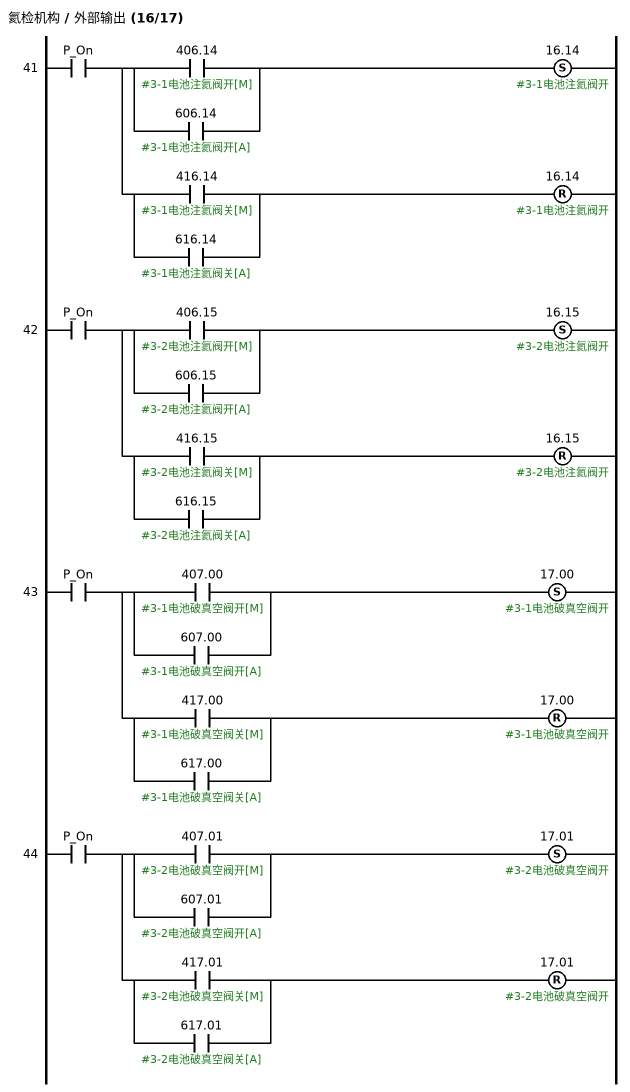
; [picture p384: 氦检机构 / 外部输出, rungs 41-44]
; rung 41
LD P_On
OUT TR0
LD 406.14  ; #3-1电池注氦阀开[M]
OR 606.14  ; #3-1电池注氦阀开[A]
ANDLD
SET 16.14  ; #3-1电池注氦阀开
LD TR0
LD 416.14  ; #3-1电池注氦阀关[M]
OR 616.14  ; #3-1电池注氦阀关[A]
ANDLD
RSET 16.14  ; #3-1电池注氦阀开
; rung 42
LD P_On
OUT TR0
LD 406.15  ; #3-2电池注氦阀开[M]
OR 606.15  ; #3-2电池注氦阀开[A]
ANDLD
SET 16.15  ; #3-2电池注氦阀开
LD TR0
LD 416.15  ; #3-2电池注氦阀关[M]
OR 616.15  ; #3-2电池注氦阀关[A]
ANDLD
RSET 16.15  ; #3-2电池注氦阀开
; rung 43
LD P_On
OUT TR0
LD 407.00  ; #3-1电池破真空阀开[M]
OR 607.00  ; #3-1电池破真空阀开[A]
ANDLD
SET 17.00  ; #3-1电池破真空阀开
LD TR0
LD 417.00  ; #3-1电池破真空阀关[M]
OR 617.00  ; #3-1电池破真空阀关[A]
ANDLD
RSET 17.00  ; #3-1电池破真空阀开
; rung 44
LD P_On
OUT TR0
LD 407.01  ; #3-2电池破真空阀开[M]
OR 607.01  ; #3-2电池破真空阀开[A]
ANDLD
SET 17.01  ; #3-2电池破真空阀开
LD TR0
LD 417.01  ; #3-2电池破真空阀关[M]
OR 617.01  ; #3-2电池破真空阀关[A]
ANDLD
RSET 17.01  ; #3-2电池破真空阀开

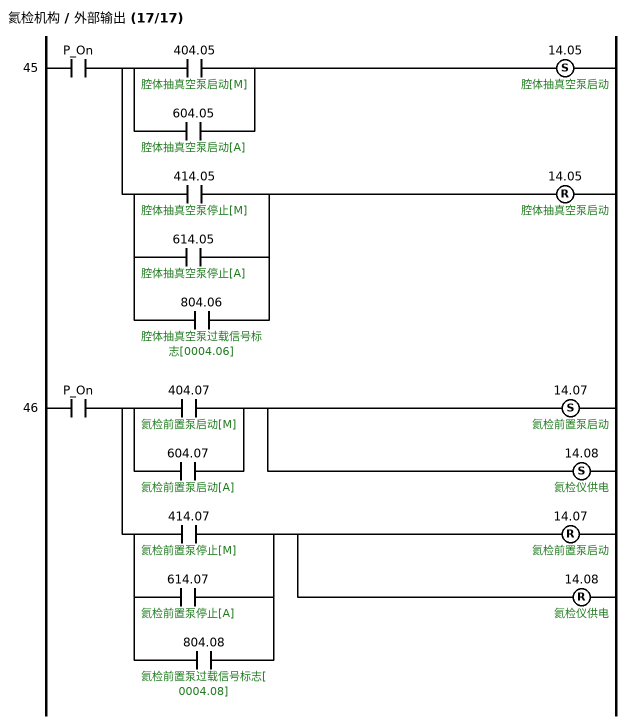
; rung 45
LD P_On
OUT TR0
LD 404.05  ; 腔体抽真空泵启动[M]
OR 604.05  ; 腔体抽真空泵启动[A]
ANDLD
SET 14.05  ; 腔体抽真空泵启动
LD TR0
LD 414.05  ; 腔体抽真空泵停止[M]
OR 614.05  ; 腔体抽真空泵停止[A]
OR 804.06  ; 腔体抽真空泵过载信号标志[0004.06]
ANDLD
RSET 14.05  ; 腔体抽真空泵启动
; rung 46
LD P_On
OUT TR0
LD 404.07  ; 氦检前置泵启动[M]
OR 604.07  ; 氦检前置泵启动[A]
ANDLD
SET 14.07  ; 氦检前置泵启动
SET 14.08  ; 氦检仪供电
LD TR0
LD 414.07  ; 氦检前置泵停止[M]
OR 614.07  ; 氦检前置泵停止[A]
OR 804.08  ; 氦检前置泵过载信号标志[0004.08]
ANDLD
RSET 14.07  ; 氦检前置泵启动
RSET 14.08  ; 氦检仪供电

### Section END
; rung 0
END(001)

## Program 出料伺服机构 (cyclic task 4)

### Section Main

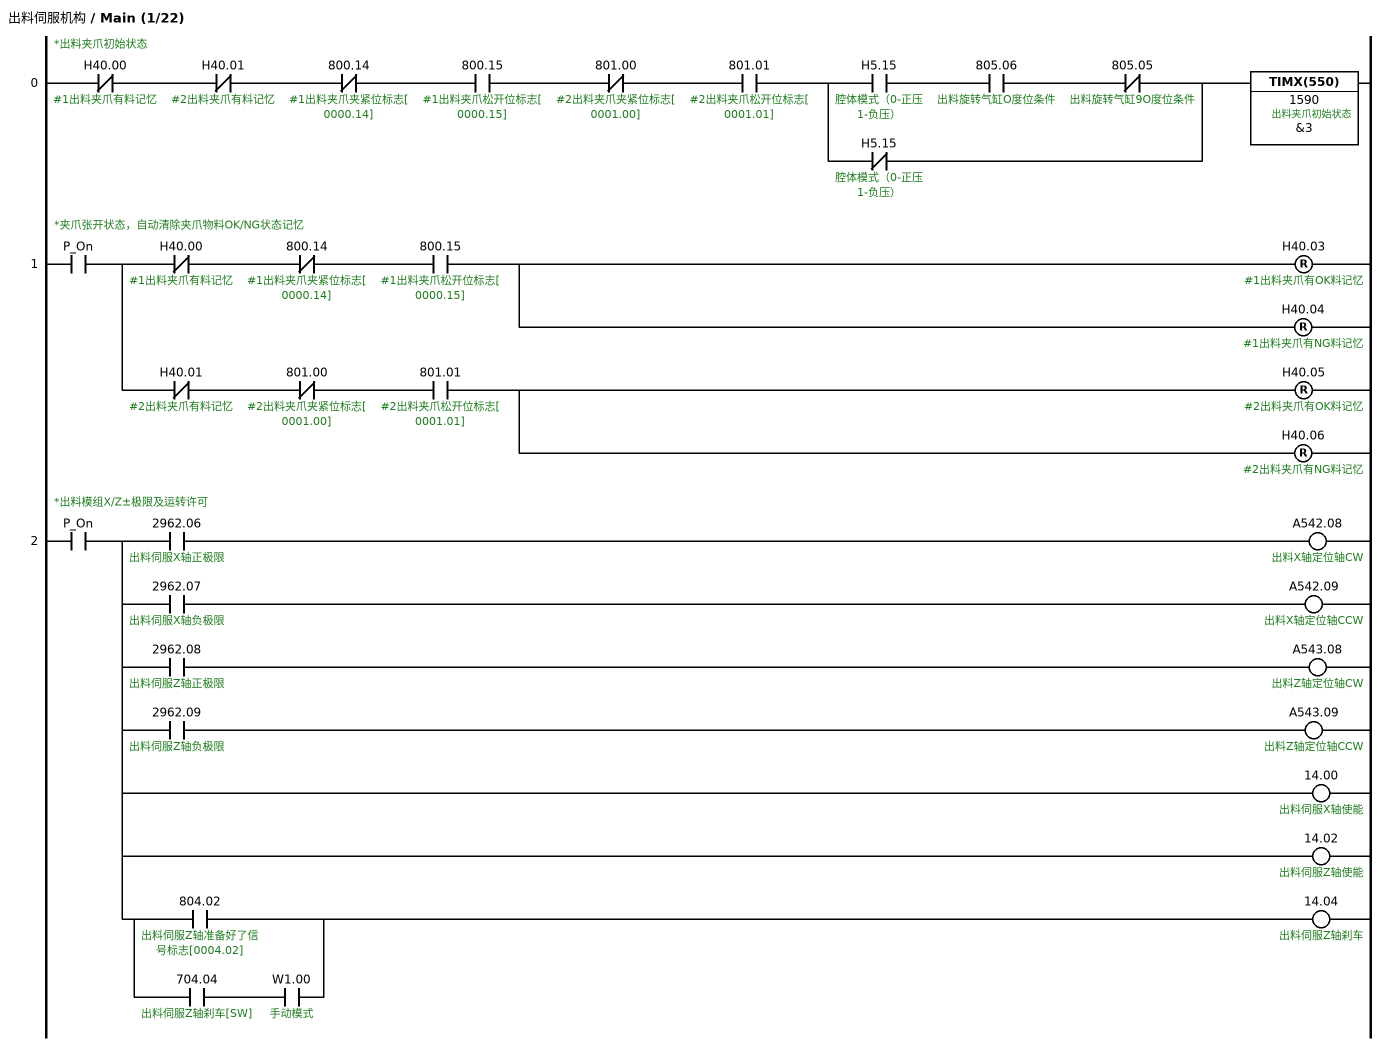
; rung 0: *出料夹爪初始状态
LDNOT H40.00  ; #1出料夹爪有料记忆
ANDNOT H40.01  ; #2出料夹爪有料记忆
ANDNOT 800.14  ; #1出料夹爪夹紧位标志[0000.14]
AND 800.15  ; #1出料夹爪松开位标志[0000.15]
ANDNOT 801.00  ; #2出料夹爪夹紧位标志[0001.00]
AND 801.01  ; #2出料夹爪松开位标志[0001.01]
LD H5.15  ; 腔体模式（0-正压 1-负压）
AND 805.06  ; 出料旋转气缸O度位条件
ANDNOT 805.05  ; 出料旋转气缸9O度位条件
ORNOT H5.15  ; 腔体模式（0-正压 1-负压）
ANDLD
TIMX(550) 1590 &3  ; 出料夹爪初始状态
; rung 1: *夹爪张开状态，自动清除夹爪物料OK/NG状态记忆
LD P_On
OUT TR0
ANDNOT H40.00  ; #1出料夹爪有料记忆
ANDNOT 800.14  ; #1出料夹爪夹紧位标志[0000.14]
AND 800.15  ; #1出料夹爪松开位标志[0000.15]
RSET H40.03  ; #1出料夹爪有OK料记忆
RSET H40.04  ; #1出料夹爪有NG料记忆
LD TR0
ANDNOT H40.01  ; #2出料夹爪有料记忆
ANDNOT 801.00  ; #2出料夹爪夹紧位标志[0001.00]
AND 801.01  ; #2出料夹爪松开位标志[0001.01]
RSET H40.05  ; #2出料夹爪有OK料记忆
RSET H40.06  ; #2出料夹爪有NG料记忆
; rung 2: *出料模组X/Z±极限及运转许可
LD P_On
OUT TR0
AND 2962.06  ; 出料伺服X轴正极限
OUT A542.08  ; 出料X轴定位轴CW
LD TR0
AND 2962.07  ; 出料伺服X轴负极限
OUT A542.09  ; 出料X轴定位轴CCW
LD TR0
AND 2962.08  ; 出料伺服Z轴正极限
OUT A543.08  ; 出料Z轴定位轴CW
LD TR0
AND 2962.09  ; 出料伺服Z轴负极限
OUT A543.09  ; 出料Z轴定位轴CCW
LD TR0
OUT 14.00  ; 出料伺服X轴使能
OUT 14.02  ; 出料伺服Z轴使能
LD 804.02  ; 出料伺服Z轴准备好了信号标志[0004.02]
LD 704.04  ; 出料伺服Z轴刹车[SW]
AND W1.00  ; 手动模式
ORLD
ANDLD
OUT 14.04  ; 出料伺服Z轴刹车

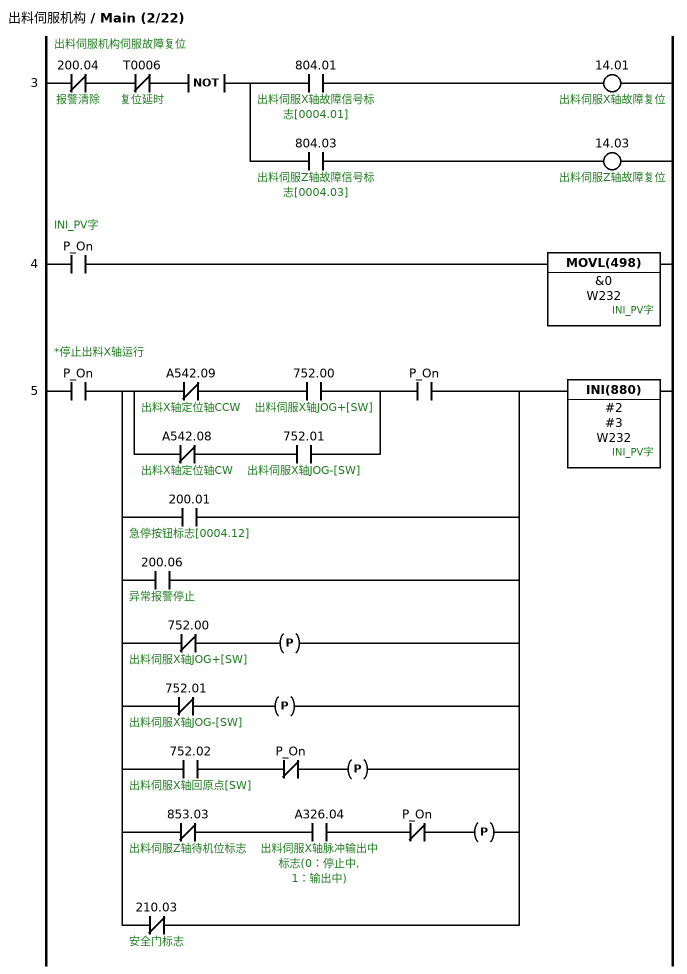
; rung 3: 出料伺服机构伺服故障复位
LDNOT 200.04  ; 报警清除
ANDNOT T0006  ; 复位延时
NOT(520)
OUT TR0
AND 804.01  ; 出料伺服X轴故障信号标志[0004.01]
OUT 14.01  ; 出料伺服X轴故障复位
LD TR0
AND 804.03  ; 出料伺服Z轴故障信号标志[0004.03]
OUT 14.03  ; 出料伺服Z轴故障复位
; rung 4: INI_PV字
LD P_On
MOVL(498) &0 W232  ; INI_PV字
; rung 5: *停止出料X轴运行
LD P_On
LDNOT A542.09  ; 出料X轴定位轴CCW
AND 752.00  ; 出料伺服X轴JOG+[SW]
LDNOT A542.08  ; 出料X轴定位轴CW
AND 752.01  ; 出料伺服X轴JOG-[SW]
ORLD
AND P_On
OR 200.01  ; 急停按钮标志[0004.12]
OR 200.06  ; 异常报警停止
LDNOT 752.00  ; 出料伺服X轴JOG+[SW]
UP(521)
ORLD
LDNOT 752.01  ; 出料伺服X轴JOG-[SW]
UP(521)
ORLD
LD 752.02  ; 出料伺服X轴回原点[SW]
ANDNOT P_On
UP(521)
ORLD
LDNOT 853.03  ; 出料伺服Z轴待机位标志
AND A326.04  ; 出料伺服X轴脉冲输出中标志(0：停止中,1：输出中)
ANDNOT P_On
UP(521)
ORLD
ORNOT 210.03  ; 安全门标志
ANDLD
INI(880) #2 #3 W232  ; INI_PV字

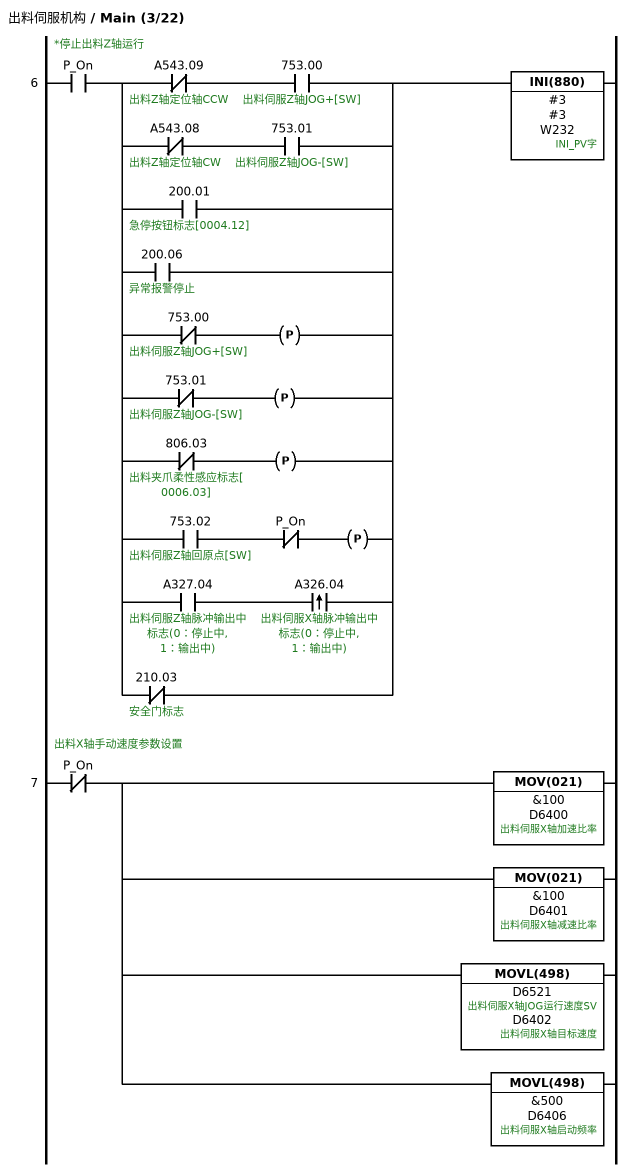
; rung 6: *停止出料Z轴运行
LD P_On
LDNOT A543.09  ; 出料Z轴定位轴CCW
AND 753.00  ; 出料伺服Z轴JOG+[SW]
LDNOT A543.08  ; 出料Z轴定位轴CW
AND 753.01  ; 出料伺服Z轴JOG-[SW]
ORLD
OR 200.01  ; 急停按钮标志[0004.12]
OR 200.06  ; 异常报警停止
LDNOT 753.00  ; 出料伺服Z轴JOG+[SW]
UP(521)
ORLD
LDNOT 753.01  ; 出料伺服Z轴JOG-[SW]
UP(521)
ORLD
LDNOT 806.03  ; 出料夹爪柔性感应标志[0006.03]
UP(521)
ORLD
LD 753.02  ; 出料伺服Z轴回原点[SW]
ANDNOT P_On
UP(521)
ORLD
LD A327.04  ; 出料伺服Z轴脉冲输出中标志(0：停止中,1：输出中)
@AND A326.04  ; 出料伺服X轴脉冲输出中标志(0：停止中,1：输出中)
ORNOT 210.03  ; 安全门标志
ORLD
ANDLD
INI(880) #3 #3 W232  ; INI_PV字
; rung 7: 出料X轴手动速度参数设置
LDNOT P_On
MOV(021) &100 D6400  ; 出料伺服X轴加速比率
MOV(021) &100 D6401  ; 出料伺服X轴减速比率
MOVL(498) D6521 D6402  ; 出料伺服X轴JOG运行速度SV, 出料伺服X轴目标速度
MOVL(498) &500 D6406  ; 出料伺服X轴启动频率

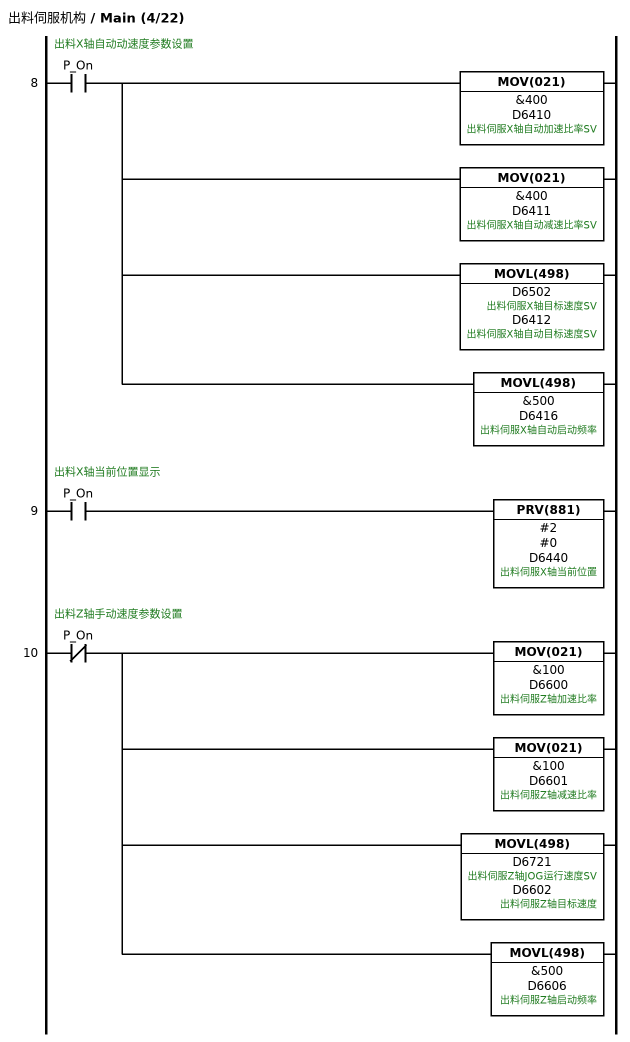
; rung 8: 出料X轴自动动速度参数设置
LD P_On
MOV(021) &400 D6410  ; 出料伺服X轴自动加速比率SV
MOV(021) &400 D6411  ; 出料伺服X轴自动减速比率SV
MOVL(498) D6502 D6412  ; 出料伺服X轴目标速度SV, 出料伺服X轴自动目标速度SV
MOVL(498) &500 D6416  ; 出料伺服X轴自动启动频率
; rung 9: 出料X轴当前位置显示
LD P_On
PRV(881) #2 #0 D6440  ; 出料伺服X轴当前位置
; rung 10: 出料Z轴手动速度参数设置
LDNOT P_On
MOV(021) &100 D6600  ; 出料伺服Z轴加速比率
MOV(021) &100 D6601  ; 出料伺服Z轴减速比率
MOVL(498) D6721 D6602  ; 出料伺服Z轴JOG运行速度SV, 出料伺服Z轴目标速度
MOVL(498) &500 D6606  ; 出料伺服Z轴启动频率

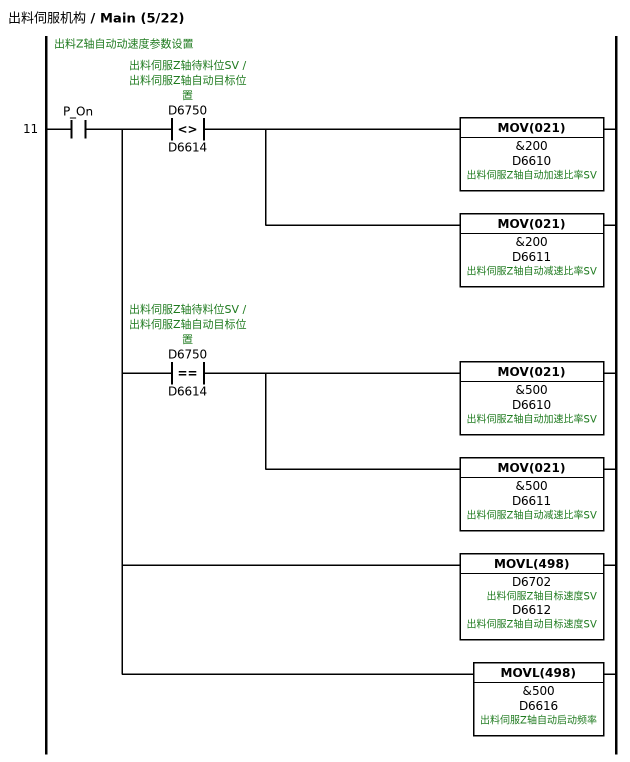
; rung 11: 出料Z轴自动动速度参数设置
LD P_On
OUT TR0
AND<>L(306) D6750 D6614  ; 出料伺服Z轴待料位SV, 出料伺服Z轴自动目标位置
MOV(021) &200 D6610  ; 出料伺服Z轴自动加速比率SV
MOV(021) &200 D6611  ; 出料伺服Z轴自动减速比率SV
LD TR0
AND=L(301) D6750 D6614  ; 出料伺服Z轴待料位SV, 出料伺服Z轴自动目标位置
MOV(021) &500 D6610  ; 出料伺服Z轴自动加速比率SV
MOV(021) &500 D6611  ; 出料伺服Z轴自动减速比率SV
LD TR0
MOVL(498) D6702 D6612  ; 出料伺服Z轴目标速度SV, 出料伺服Z轴自动目标速度SV
MOVL(498) &500 D6616  ; 出料伺服Z轴自动启动频率

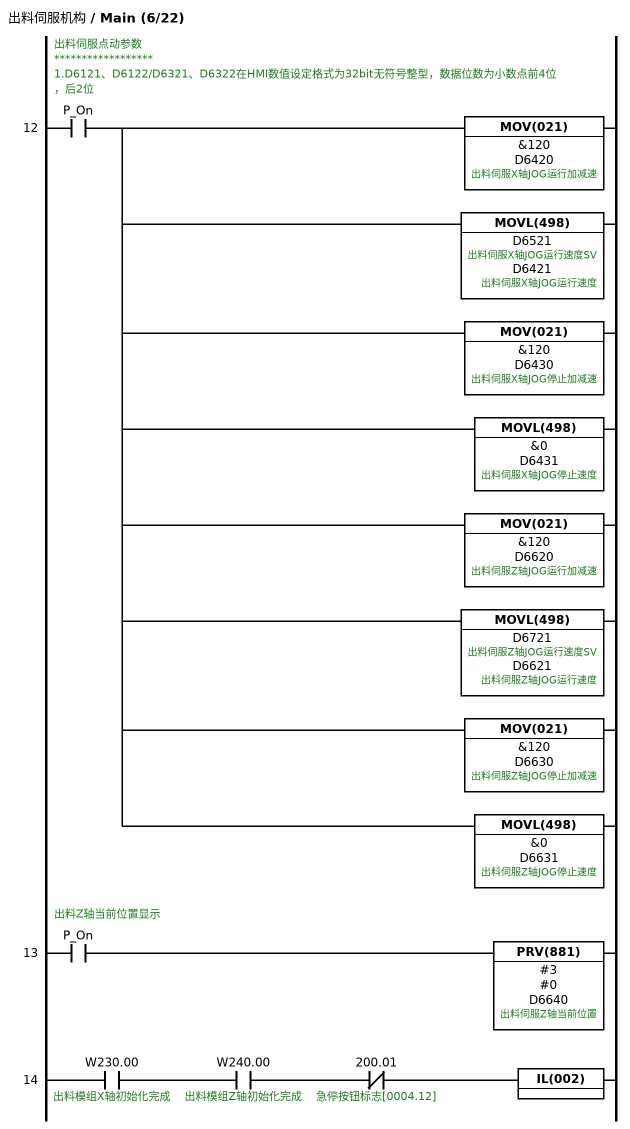
; rung 12: 出料伺服点动参数 / ****************** / 1.D6121、D6122/D6321、D6322在HMI数值设定格式为32bit无符号整型，数据位数为小数点前4位，后2位
LD P_On
MOV(021) &120 D6420  ; 出料伺服X轴JOG运行加减速
MOVL(498) D6521 D6421  ; 出料伺服X轴JOG运行速度SV, 出料伺服X轴JOG运行速度
MOV(021) &120 D6430  ; 出料伺服X轴JOG停止加减速
MOVL(498) &0 D6431  ; 出料伺服X轴JOG停止速度
MOV(021) &120 D6620  ; 出料伺服Z轴JOG运行加减速
MOVL(498) D6721 D6621  ; 出料伺服Z轴JOG运行速度SV, 出料伺服Z轴JOG运行速度
MOV(021) &120 D6630  ; 出料伺服Z轴JOG停止加减速
MOVL(498) &0 D6631  ; 出料伺服Z轴JOG停止速度
; rung 13: 出料Z轴当前位置显示
LD P_On
PRV(881) #3 #0 D6640  ; 出料伺服Z轴当前位置
; rung 14
LD W230.00  ; 出料模组X轴初始化完成
AND W240.00  ; 出料模组Z轴初始化完成
ANDNOT 200.01  ; 急停按钮标志[0004.12]
IL(002)

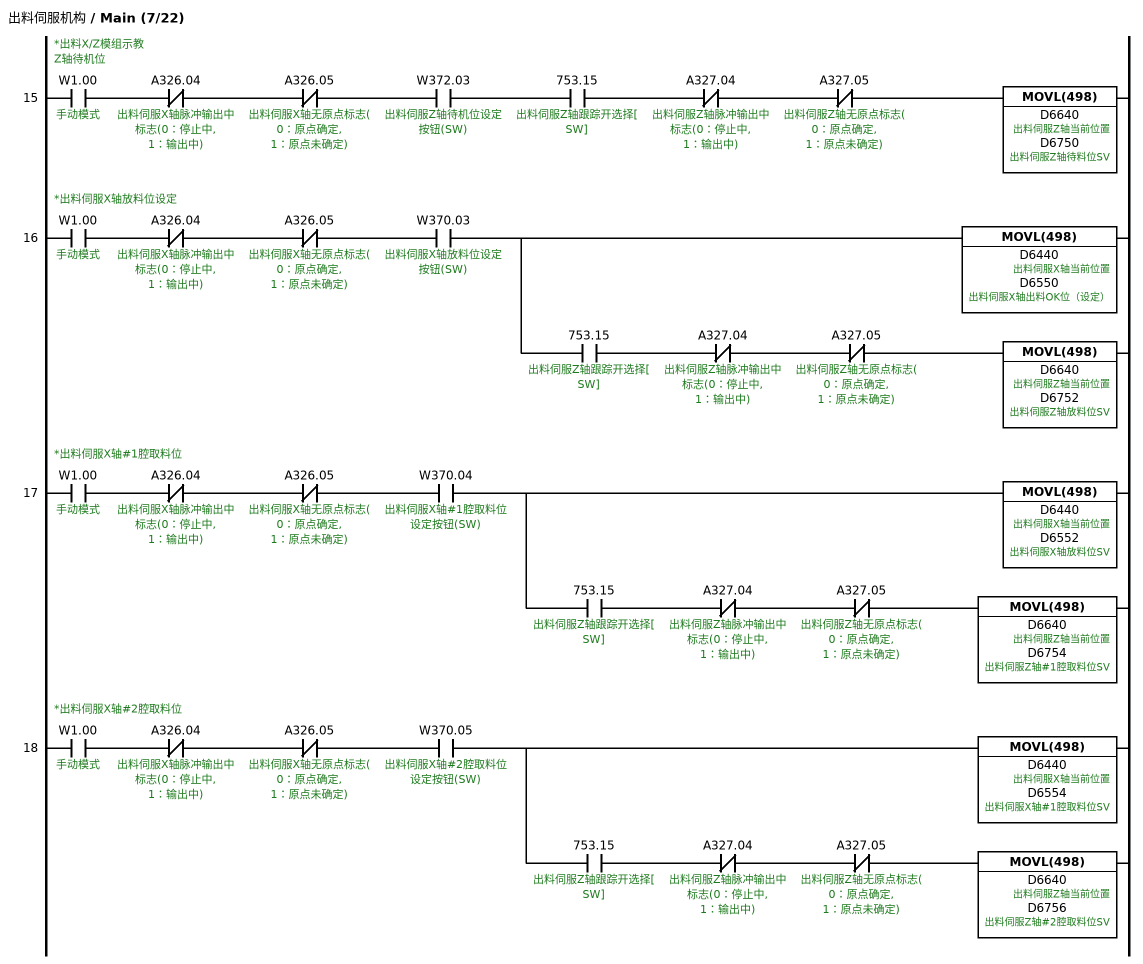
; rung 15: *出料X/Z模组示教 / Z轴待机位
LD W1.00  ; 手动模式
ANDNOT A326.04  ; 出料伺服X轴脉冲输出中标志(0：停止中,1：输出中)
ANDNOT A326.05  ; 出料伺服X轴无原点标志(0：原点确定,1：原点未确定)
AND W372.03  ; 出料伺服Z轴待机位设定按钮(SW)
AND 753.15  ; 出料伺服Z轴跟踪开选择[SW]
ANDNOT A327.04  ; 出料伺服Z轴脉冲输出中标志(0：停止中,1：输出中)
ANDNOT A327.05  ; 出料伺服Z轴无原点标志(0：原点确定,1：原点未确定)
MOVL(498) D6640 D6750  ; 出料伺服Z轴当前位置, 出料伺服Z轴待料位SV
; rung 16: *出料伺服X轴放料位设定
LD W1.00  ; 手动模式
ANDNOT A326.04  ; 出料伺服X轴脉冲输出中标志(0：停止中,1：输出中)
ANDNOT A326.05  ; 出料伺服X轴无原点标志(0：原点确定,1：原点未确定)
AND W370.03  ; 出料伺服X轴放料位设定按钮(SW)
MOVL(498) D6440 D6550  ; 出料伺服X轴当前位置, 出料伺服X轴出料OK位（设定）
AND 753.15  ; 出料伺服Z轴跟踪开选择[SW]
ANDNOT A327.04  ; 出料伺服Z轴脉冲输出中标志(0：停止中,1：输出中)
ANDNOT A327.05  ; 出料伺服Z轴无原点标志(0：原点确定,1：原点未确定)
MOVL(498) D6640 D6752  ; 出料伺服Z轴当前位置, 出料伺服Z轴放料位SV
; rung 17: *出料伺服X轴#1腔取料位
LD W1.00  ; 手动模式
ANDNOT A326.04  ; 出料伺服X轴脉冲输出中标志(0：停止中,1：输出中)
ANDNOT A326.05  ; 出料伺服X轴无原点标志(0：原点确定,1：原点未确定)
AND W370.04  ; 出料伺服X轴#1腔取料位设定按钮(SW)
MOVL(498) D6440 D6552  ; 出料伺服X轴当前位置, 出料伺服X轴放料位SV
AND 753.15  ; 出料伺服Z轴跟踪开选择[SW]
ANDNOT A327.04  ; 出料伺服Z轴脉冲输出中标志(0：停止中,1：输出中)
ANDNOT A327.05  ; 出料伺服Z轴无原点标志(0：原点确定,1：原点未确定)
MOVL(498) D6640 D6754  ; 出料伺服Z轴当前位置, 出料伺服Z轴#1腔取料位SV
; rung 18: *出料伺服X轴#2腔取料位
LD W1.00  ; 手动模式
ANDNOT A326.04  ; 出料伺服X轴脉冲输出中标志(0：停止中,1：输出中)
ANDNOT A326.05  ; 出料伺服X轴无原点标志(0：原点确定,1：原点未确定)
AND W370.05  ; 出料伺服X轴#2腔取料位设定按钮(SW)
MOVL(498) D6440 D6554  ; 出料伺服X轴当前位置, 出料伺服X轴#1腔取料位SV
AND 753.15  ; 出料伺服Z轴跟踪开选择[SW]
ANDNOT A327.04  ; 出料伺服Z轴脉冲输出中标志(0：停止中,1：输出中)
ANDNOT A327.05  ; 出料伺服Z轴无原点标志(0：原点确定,1：原点未确定)
MOVL(498) D6640 D6756  ; 出料伺服Z轴当前位置, 出料伺服Z轴#2腔取料位SV

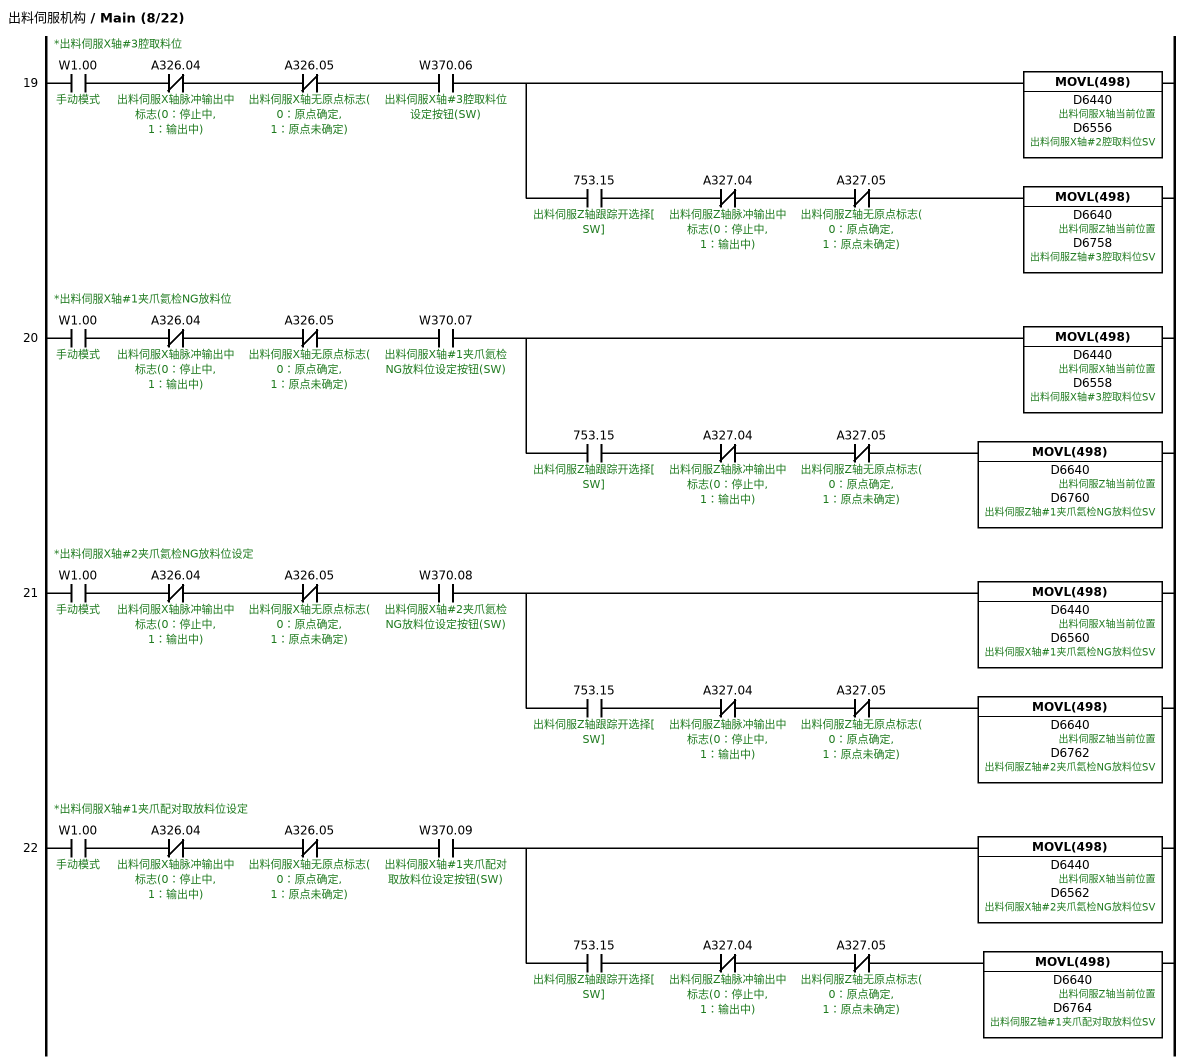
; rung 19: *出料伺服X轴#3腔取料位
LD W1.00  ; 手动模式
ANDNOT A326.04  ; 出料伺服X轴脉冲输出中标志(0：停止中,1：输出中)
ANDNOT A326.05  ; 出料伺服X轴无原点标志(0：原点确定,1：原点未确定)
AND W370.06  ; 出料伺服X轴#3腔取料位设定按钮(SW)
MOVL(498) D6440 D6556  ; 出料伺服X轴当前位置, 出料伺服X轴#2腔取料位SV
AND 753.15  ; 出料伺服Z轴跟踪开选择[SW]
ANDNOT A327.04  ; 出料伺服Z轴脉冲输出中标志(0：停止中,1：输出中)
ANDNOT A327.05  ; 出料伺服Z轴无原点标志(0：原点确定,1：原点未确定)
MOVL(498) D6640 D6758  ; 出料伺服Z轴当前位置, 出料伺服Z轴#3腔取料位SV
; rung 20: *出料伺服X轴#1夹爪氦检NG放料位
LD W1.00  ; 手动模式
ANDNOT A326.04  ; 出料伺服X轴脉冲输出中标志(0：停止中,1：输出中)
ANDNOT A326.05  ; 出料伺服X轴无原点标志(0：原点确定,1：原点未确定)
AND W370.07  ; 出料伺服X轴#1夹爪氦检NG放料位设定按钮(SW)
MOVL(498) D6440 D6558  ; 出料伺服X轴当前位置, 出料伺服X轴#3腔取料位SV
AND 753.15  ; 出料伺服Z轴跟踪开选择[SW]
ANDNOT A327.04  ; 出料伺服Z轴脉冲输出中标志(0：停止中,1：输出中)
ANDNOT A327.05  ; 出料伺服Z轴无原点标志(0：原点确定,1：原点未确定)
MOVL(498) D6640 D6760  ; 出料伺服Z轴当前位置, 出料伺服Z轴#1夹爪氦检NG放料位SV
; rung 21: *出料伺服X轴#2夹爪氦检NG放料位设定
LD W1.00  ; 手动模式
ANDNOT A326.04  ; 出料伺服X轴脉冲输出中标志(0：停止中,1：输出中)
ANDNOT A326.05  ; 出料伺服X轴无原点标志(0：原点确定,1：原点未确定)
AND W370.08  ; 出料伺服X轴#2夹爪氦检NG放料位设定按钮(SW)
MOVL(498) D6440 D6560  ; 出料伺服X轴当前位置, 出料伺服X轴#1夹爪氦检NG放料位SV
AND 753.15  ; 出料伺服Z轴跟踪开选择[SW]
ANDNOT A327.04  ; 出料伺服Z轴脉冲输出中标志(0：停止中,1：输出中)
ANDNOT A327.05  ; 出料伺服Z轴无原点标志(0：原点确定,1：原点未确定)
MOVL(498) D6640 D6762  ; 出料伺服Z轴当前位置, 出料伺服Z轴#2夹爪氦检NG放料位SV
; rung 22: *出料伺服X轴#1夹爪配对取放料位设定
LD W1.00  ; 手动模式
ANDNOT A326.04  ; 出料伺服X轴脉冲输出中标志(0：停止中,1：输出中)
ANDNOT A326.05  ; 出料伺服X轴无原点标志(0：原点确定,1：原点未确定)
AND W370.09  ; 出料伺服X轴#1夹爪配对取放料位设定按钮(SW)
MOVL(498) D6440 D6562  ; 出料伺服X轴当前位置, 出料伺服X轴#2夹爪氦检NG放料位SV
AND 753.15  ; 出料伺服Z轴跟踪开选择[SW]
ANDNOT A327.04  ; 出料伺服Z轴脉冲输出中标志(0：停止中,1：输出中)
ANDNOT A327.05  ; 出料伺服Z轴无原点标志(0：原点确定,1：原点未确定)
MOVL(498) D6640 D6764  ; 出料伺服Z轴当前位置, 出料伺服Z轴#1夹爪配对取放料位SV

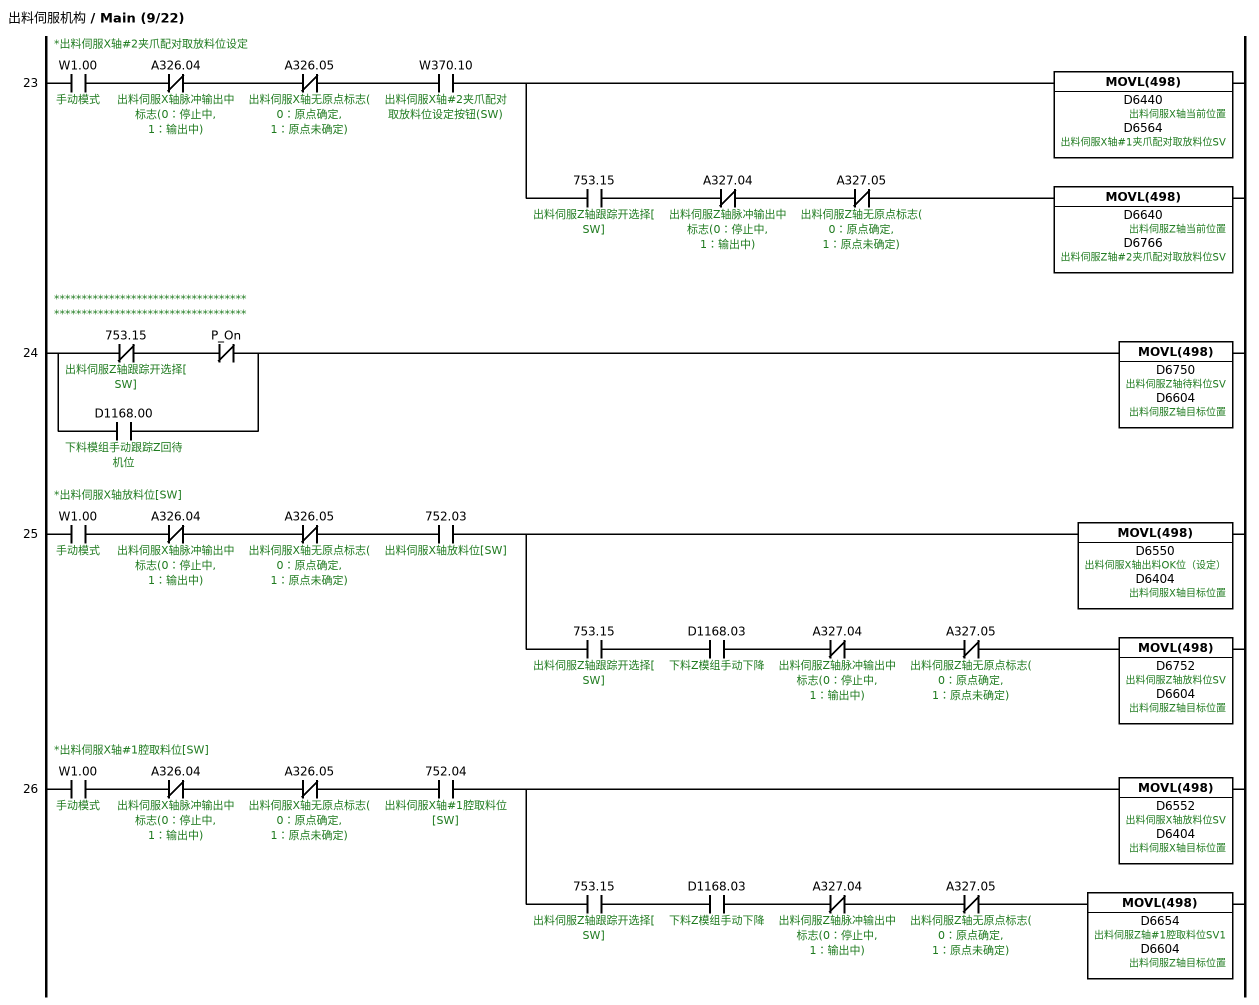
; rung 23: *出料伺服X轴#2夹爪配对取放料位设定
LD W1.00  ; 手动模式
ANDNOT A326.04  ; 出料伺服X轴脉冲输出中标志(0：停止中,1：输出中)
ANDNOT A326.05  ; 出料伺服X轴无原点标志(0：原点确定,1：原点未确定)
AND W370.10  ; 出料伺服X轴#2夹爪配对取放料位设定按钮(SW)
MOVL(498) D6440 D6564  ; 出料伺服X轴当前位置, 出料伺服X轴#1夹爪配对取放料位SV
AND 753.15  ; 出料伺服Z轴跟踪开选择[SW]
ANDNOT A327.04  ; 出料伺服Z轴脉冲输出中标志(0：停止中,1：输出中)
ANDNOT A327.05  ; 出料伺服Z轴无原点标志(0：原点确定,1：原点未确定)
MOVL(498) D6640 D6766  ; 出料伺服Z轴当前位置, 出料伺服Z轴#2夹爪配对取放料位SV
; rung 24: *********************************** / ***********************************
LDNOT 753.15  ; 出料伺服Z轴跟踪开选择[SW]
ANDNOT P_On
OR D1168.00  ; 下料模组手动跟踪Z回待机位
MOVL(498) D6750 D6604  ; 出料伺服Z轴待料位SV, 出料伺服Z轴目标位置
; rung 25: *出料伺服X轴放料位[SW]
LD W1.00  ; 手动模式
ANDNOT A326.04  ; 出料伺服X轴脉冲输出中标志(0：停止中,1：输出中)
ANDNOT A326.05  ; 出料伺服X轴无原点标志(0：原点确定,1：原点未确定)
AND 752.03  ; 出料伺服X轴放料位[SW]
MOVL(498) D6550 D6404  ; 出料伺服X轴出料OK位（设定）, 出料伺服X轴目标位置
AND 753.15  ; 出料伺服Z轴跟踪开选择[SW]
AND D1168.03  ; 下料Z模组手动下降
ANDNOT A327.04  ; 出料伺服Z轴脉冲输出中标志(0：停止中,1：输出中)
ANDNOT A327.05  ; 出料伺服Z轴无原点标志(0：原点确定,1：原点未确定)
MOVL(498) D6752 D6604  ; 出料伺服Z轴放料位SV, 出料伺服Z轴目标位置
; rung 26: *出料伺服X轴#1腔取料位[SW]
LD W1.00  ; 手动模式
ANDNOT A326.04  ; 出料伺服X轴脉冲输出中标志(0：停止中,1：输出中)
ANDNOT A326.05  ; 出料伺服X轴无原点标志(0：原点确定,1：原点未确定)
AND 752.04  ; 出料伺服X轴#1腔取料位[SW]
MOVL(498) D6552 D6404  ; 出料伺服X轴放料位SV, 出料伺服X轴目标位置
AND 753.15  ; 出料伺服Z轴跟踪开选择[SW]
AND D1168.03  ; 下料Z模组手动下降
ANDNOT A327.04  ; 出料伺服Z轴脉冲输出中标志(0：停止中,1：输出中)
ANDNOT A327.05  ; 出料伺服Z轴无原点标志(0：原点确定,1：原点未确定)
MOVL(498) D6654 D6604  ; 出料伺服Z轴#1腔取料位SV1, 出料伺服Z轴目标位置

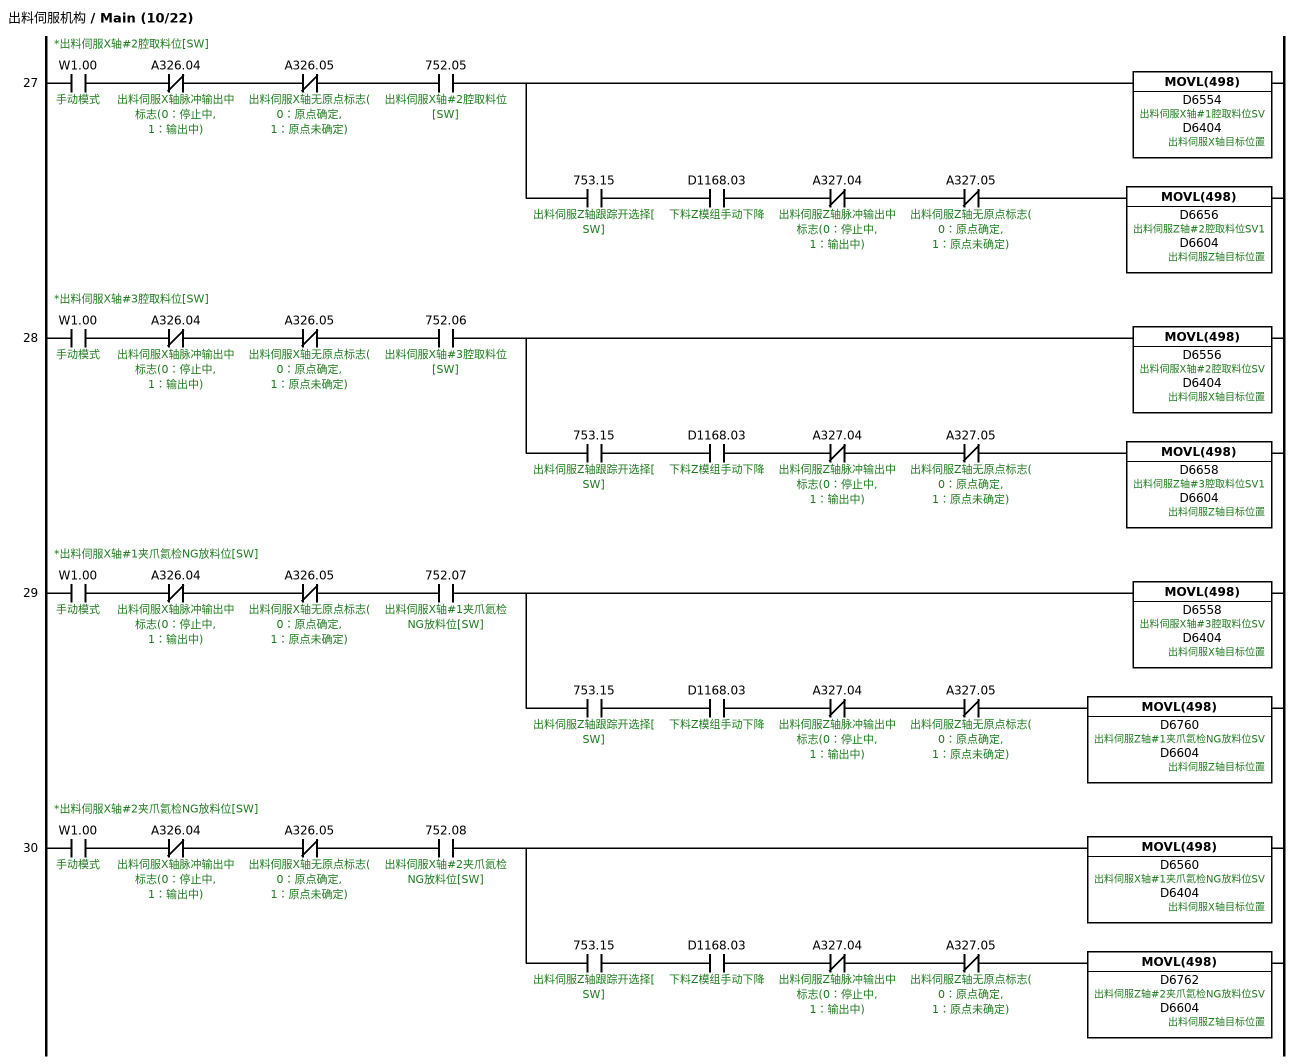
; rung 27: *出料伺服X轴#2腔取料位[SW]
LD W1.00  ; 手动模式
ANDNOT A326.04  ; 出料伺服X轴脉冲输出中标志(0：停止中,1：输出中)
ANDNOT A326.05  ; 出料伺服X轴无原点标志(0：原点确定,1：原点未确定)
AND 752.05  ; 出料伺服X轴#2腔取料位[SW]
MOVL(498) D6554 D6404  ; 出料伺服X轴#1腔取料位SV, 出料伺服X轴目标位置
AND 753.15  ; 出料伺服Z轴跟踪开选择[SW]
AND D1168.03  ; 下料Z模组手动下降
ANDNOT A327.04  ; 出料伺服Z轴脉冲输出中标志(0：停止中,1：输出中)
ANDNOT A327.05  ; 出料伺服Z轴无原点标志(0：原点确定,1：原点未确定)
MOVL(498) D6656 D6604  ; 出料伺服Z轴#2腔取料位SV1, 出料伺服Z轴目标位置
; rung 28: *出料伺服X轴#3腔取料位[SW]
LD W1.00  ; 手动模式
ANDNOT A326.04  ; 出料伺服X轴脉冲输出中标志(0：停止中,1：输出中)
ANDNOT A326.05  ; 出料伺服X轴无原点标志(0：原点确定,1：原点未确定)
AND 752.06  ; 出料伺服X轴#3腔取料位[SW]
MOVL(498) D6556 D6404  ; 出料伺服X轴#2腔取料位SV, 出料伺服X轴目标位置
AND 753.15  ; 出料伺服Z轴跟踪开选择[SW]
AND D1168.03  ; 下料Z模组手动下降
ANDNOT A327.04  ; 出料伺服Z轴脉冲输出中标志(0：停止中,1：输出中)
ANDNOT A327.05  ; 出料伺服Z轴无原点标志(0：原点确定,1：原点未确定)
MOVL(498) D6658 D6604  ; 出料伺服Z轴#3腔取料位SV1, 出料伺服Z轴目标位置
; rung 29: *出料伺服X轴#1夹爪氦检NG放料位[SW]
LD W1.00  ; 手动模式
ANDNOT A326.04  ; 出料伺服X轴脉冲输出中标志(0：停止中,1：输出中)
ANDNOT A326.05  ; 出料伺服X轴无原点标志(0：原点确定,1：原点未确定)
AND 752.07  ; 出料伺服X轴#1夹爪氦检NG放料位[SW]
MOVL(498) D6558 D6404  ; 出料伺服X轴#3腔取料位SV, 出料伺服X轴目标位置
AND 753.15  ; 出料伺服Z轴跟踪开选择[SW]
AND D1168.03  ; 下料Z模组手动下降
ANDNOT A327.04  ; 出料伺服Z轴脉冲输出中标志(0：停止中,1：输出中)
ANDNOT A327.05  ; 出料伺服Z轴无原点标志(0：原点确定,1：原点未确定)
MOVL(498) D6760 D6604  ; 出料伺服Z轴#1夹爪氦检NG放料位SV, 出料伺服Z轴目标位置
; rung 30: *出料伺服X轴#2夹爪氦检NG放料位[SW]
LD W1.00  ; 手动模式
ANDNOT A326.04  ; 出料伺服X轴脉冲输出中标志(0：停止中,1：输出中)
ANDNOT A326.05  ; 出料伺服X轴无原点标志(0：原点确定,1：原点未确定)
AND 752.08  ; 出料伺服X轴#2夹爪氦检NG放料位[SW]
MOVL(498) D6560 D6404  ; 出料伺服X轴#1夹爪氦检NG放料位SV, 出料伺服X轴目标位置
AND 753.15  ; 出料伺服Z轴跟踪开选择[SW]
AND D1168.03  ; 下料Z模组手动下降
ANDNOT A327.04  ; 出料伺服Z轴脉冲输出中标志(0：停止中,1：输出中)
ANDNOT A327.05  ; 出料伺服Z轴无原点标志(0：原点确定,1：原点未确定)
MOVL(498) D6762 D6604  ; 出料伺服Z轴#2夹爪氦检NG放料位SV, 出料伺服Z轴目标位置

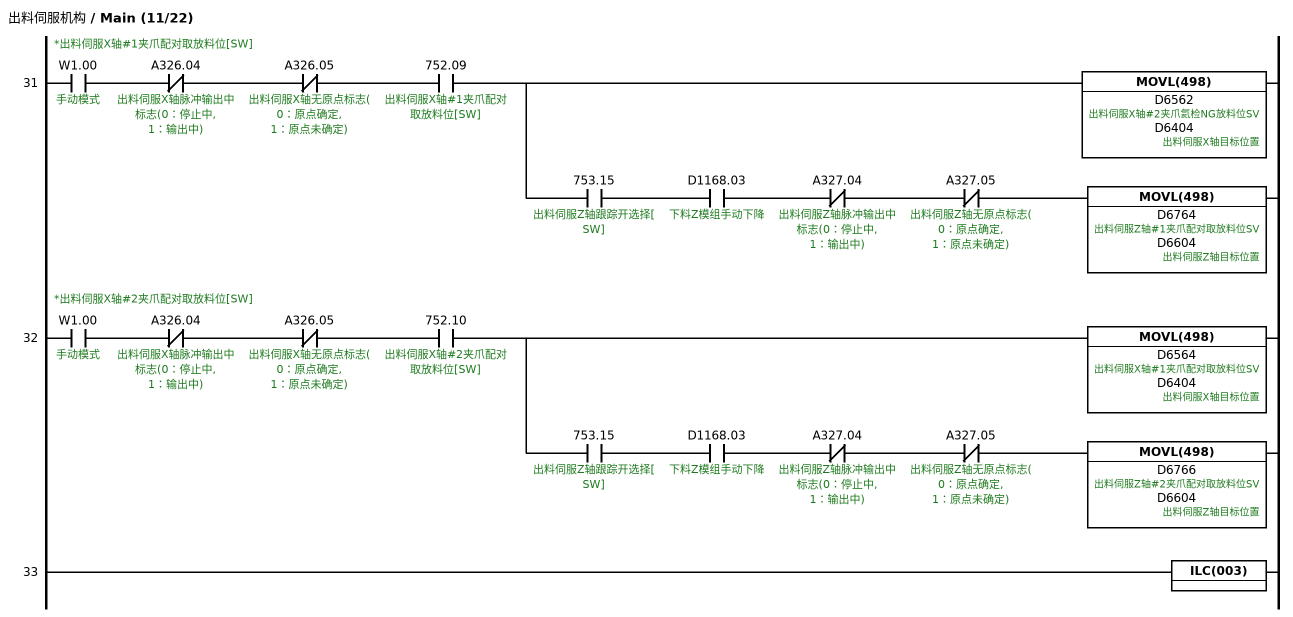
; rung 31: *出料伺服X轴#1夹爪配对取放料位[SW]
LD W1.00  ; 手动模式
ANDNOT A326.04  ; 出料伺服X轴脉冲输出中标志(0：停止中,1：输出中)
ANDNOT A326.05  ; 出料伺服X轴无原点标志(0：原点确定,1：原点未确定)
AND 752.09  ; 出料伺服X轴#1夹爪配对取放料位[SW]
MOVL(498) D6562 D6404  ; 出料伺服X轴#2夹爪氦检NG放料位SV, 出料伺服X轴目标位置
AND 753.15  ; 出料伺服Z轴跟踪开选择[SW]
AND D1168.03  ; 下料Z模组手动下降
ANDNOT A327.04  ; 出料伺服Z轴脉冲输出中标志(0：停止中,1：输出中)
ANDNOT A327.05  ; 出料伺服Z轴无原点标志(0：原点确定,1：原点未确定)
MOVL(498) D6764 D6604  ; 出料伺服Z轴#1夹爪配对取放料位SV, 出料伺服Z轴目标位置
; rung 32: *出料伺服X轴#2夹爪配对取放料位[SW]
LD W1.00  ; 手动模式
ANDNOT A326.04  ; 出料伺服X轴脉冲输出中标志(0：停止中,1：输出中)
ANDNOT A326.05  ; 出料伺服X轴无原点标志(0：原点确定,1：原点未确定)
AND 752.10  ; 出料伺服X轴#2夹爪配对取放料位[SW]
MOVL(498) D6564 D6404  ; 出料伺服X轴#1夹爪配对取放料位SV, 出料伺服X轴目标位置
AND 753.15  ; 出料伺服Z轴跟踪开选择[SW]
AND D1168.03  ; 下料Z模组手动下降
ANDNOT A327.04  ; 出料伺服Z轴脉冲输出中标志(0：停止中,1：输出中)
ANDNOT A327.05  ; 出料伺服Z轴无原点标志(0：原点确定,1：原点未确定)
MOVL(498) D6766 D6604  ; 出料伺服Z轴#2夹爪配对取放料位SV, 出料伺服Z轴目标位置
; rung 33
ILC(003)

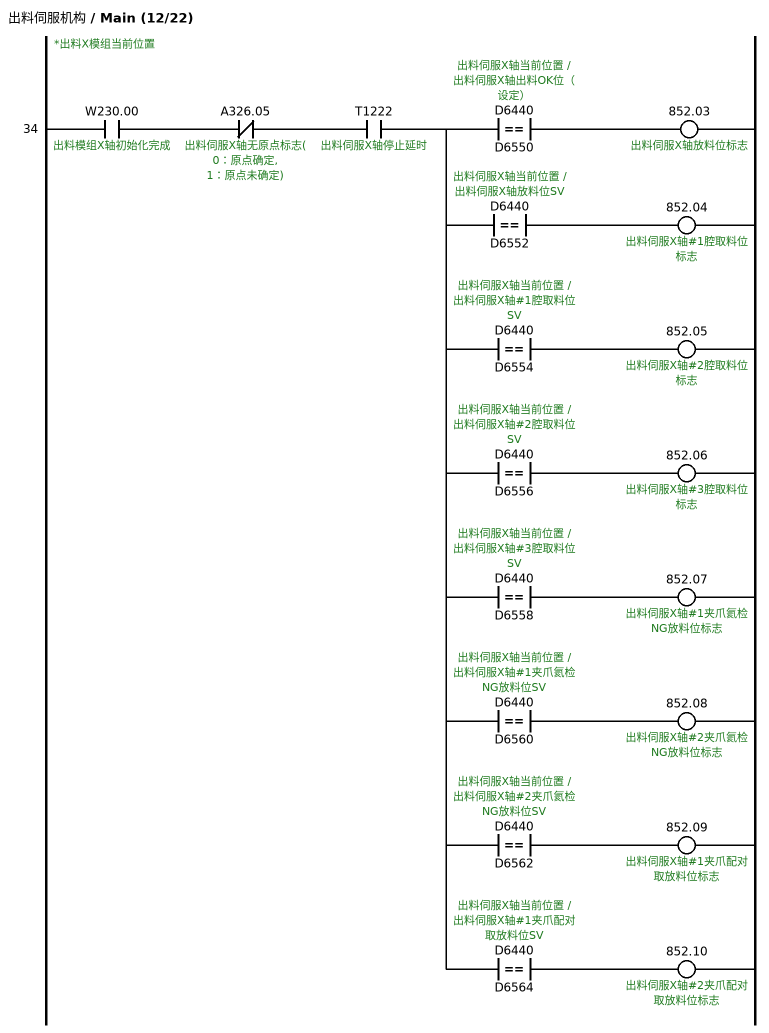
; rung 34: *出料X模组当前位置
LD W230.00  ; 出料模组X轴初始化完成
ANDNOT A326.05  ; 出料伺服X轴无原点标志(0：原点确定,1：原点未确定)
AND T1222  ; 出料伺服X轴停止延时
OUT TR0
AND=SL(303) D6440 D6550  ; 出料伺服X轴当前位置, 出料伺服X轴出料OK位（设定）
OUT 852.03  ; 出料伺服X轴放料位标志
LD TR0
AND=SL(303) D6440 D6552  ; 出料伺服X轴当前位置, 出料伺服X轴放料位SV
OUT 852.04  ; 出料伺服X轴#1腔取料位标志
LD TR0
AND=SL(303) D6440 D6554  ; 出料伺服X轴当前位置, 出料伺服X轴#1腔取料位SV
OUT 852.05  ; 出料伺服X轴#2腔取料位标志
LD TR0
AND=SL(303) D6440 D6556  ; 出料伺服X轴当前位置, 出料伺服X轴#2腔取料位SV
OUT 852.06  ; 出料伺服X轴#3腔取料位标志
LD TR0
AND=SL(303) D6440 D6558  ; 出料伺服X轴当前位置, 出料伺服X轴#3腔取料位SV
OUT 852.07  ; 出料伺服X轴#1夹爪氦检NG放料位标志
LD TR0
AND=SL(303) D6440 D6560  ; 出料伺服X轴当前位置, 出料伺服X轴#1夹爪氦检NG放料位SV
OUT 852.08  ; 出料伺服X轴#2夹爪氦检NG放料位标志
LD TR0
AND=SL(303) D6440 D6562  ; 出料伺服X轴当前位置, 出料伺服X轴#2夹爪氦检NG放料位SV
OUT 852.09  ; 出料伺服X轴#1夹爪配对取放料位标志
LD TR0
AND=SL(303) D6440 D6564  ; 出料伺服X轴当前位置, 出料伺服X轴#1夹爪配对取放料位SV
OUT 852.10  ; 出料伺服X轴#2夹爪配对取放料位标志

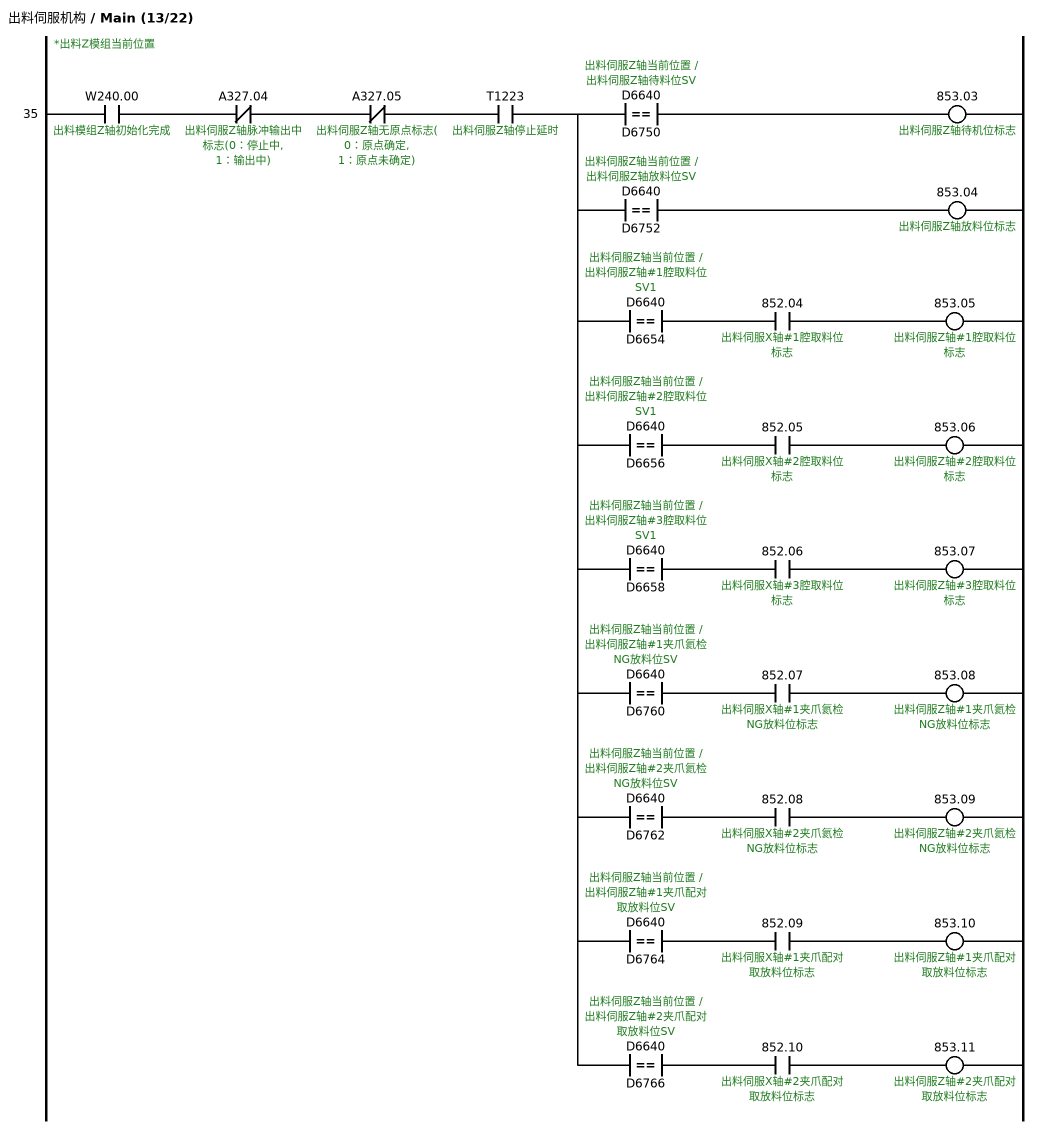
; rung 35: *出料Z模组当前位置
LD W240.00  ; 出料模组Z轴初始化完成
ANDNOT A327.04  ; 出料伺服Z轴脉冲输出中标志(0：停止中,1：输出中)
ANDNOT A327.05  ; 出料伺服Z轴无原点标志(0：原点确定,1：原点未确定)
AND T1223  ; 出料伺服Z轴停止延时
OUT TR0
AND=SL(303) D6640 D6750  ; 出料伺服Z轴当前位置, 出料伺服Z轴待料位SV
OUT 853.03  ; 出料伺服Z轴待机位标志
LD TR0
AND=SL(303) D6640 D6752  ; 出料伺服Z轴当前位置, 出料伺服Z轴放料位SV
OUT 853.04  ; 出料伺服Z轴放料位标志
LD TR0
AND=SL(303) D6640 D6654  ; 出料伺服Z轴当前位置, 出料伺服Z轴#1腔取料位SV1
AND 852.04  ; 出料伺服X轴#1腔取料位标志
OUT 853.05  ; 出料伺服Z轴#1腔取料位标志
LD TR0
AND=SL(303) D6640 D6656  ; 出料伺服Z轴当前位置, 出料伺服Z轴#2腔取料位SV1
AND 852.05  ; 出料伺服X轴#2腔取料位标志
OUT 853.06  ; 出料伺服Z轴#2腔取料位标志
LD TR0
AND=SL(303) D6640 D6658  ; 出料伺服Z轴当前位置, 出料伺服Z轴#3腔取料位SV1
AND 852.06  ; 出料伺服X轴#3腔取料位标志
OUT 853.07  ; 出料伺服Z轴#3腔取料位标志
LD TR0
AND=SL(303) D6640 D6760  ; 出料伺服Z轴当前位置, 出料伺服Z轴#1夹爪氦检NG放料位SV
AND 852.07  ; 出料伺服X轴#1夹爪氦检NG放料位标志
OUT 853.08  ; 出料伺服Z轴#1夹爪氦检NG放料位标志
LD TR0
AND=SL(303) D6640 D6762  ; 出料伺服Z轴当前位置, 出料伺服Z轴#2夹爪氦检NG放料位SV
AND 852.08  ; 出料伺服X轴#2夹爪氦检NG放料位标志
OUT 853.09  ; 出料伺服Z轴#2夹爪氦检NG放料位标志
LD TR0
AND=SL(303) D6640 D6764  ; 出料伺服Z轴当前位置, 出料伺服Z轴#1夹爪配对取放料位SV
AND 852.09  ; 出料伺服X轴#1夹爪配对取放料位标志
OUT 853.10  ; 出料伺服Z轴#1夹爪配对取放料位标志
LD TR0
AND=SL(303) D6640 D6766  ; 出料伺服Z轴当前位置, 出料伺服Z轴#2夹爪配对取放料位SV
AND 852.10  ; 出料伺服X轴#2夹爪配对取放料位标志
OUT 853.11  ; 出料伺服Z轴#2夹爪配对取放料位标志

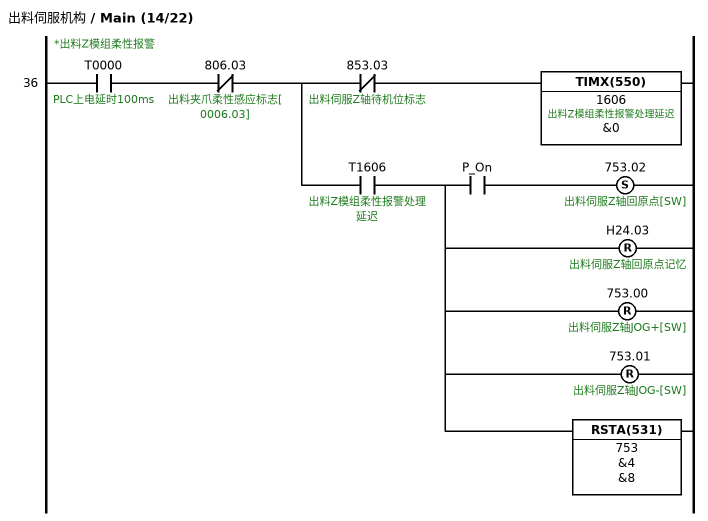
; rung 36: *出料Z模组柔性报警
LD T0000  ; PLC上电延时100ms
ANDNOT 806.03  ; 出料夹爪柔性感应标志[0006.03]
OUT TR0
ANDNOT 853.03  ; 出料伺服Z轴待机位标志
TIMX(550) 1606 &0  ; 出料Z模组柔性报警处理延迟
LD TR0
AND T1606  ; 出料Z模组柔性报警处理延迟
OUT TR0
AND P_On
SET 753.02  ; 出料伺服Z轴回原点[SW]
LD TR0
RSET H24.03  ; 出料伺服Z轴回原点记忆
RSET 753.00  ; 出料伺服Z轴JOG+[SW]
RSET 753.01  ; 出料伺服Z轴JOG-[SW]
RSTA(531) 753 &4 &8

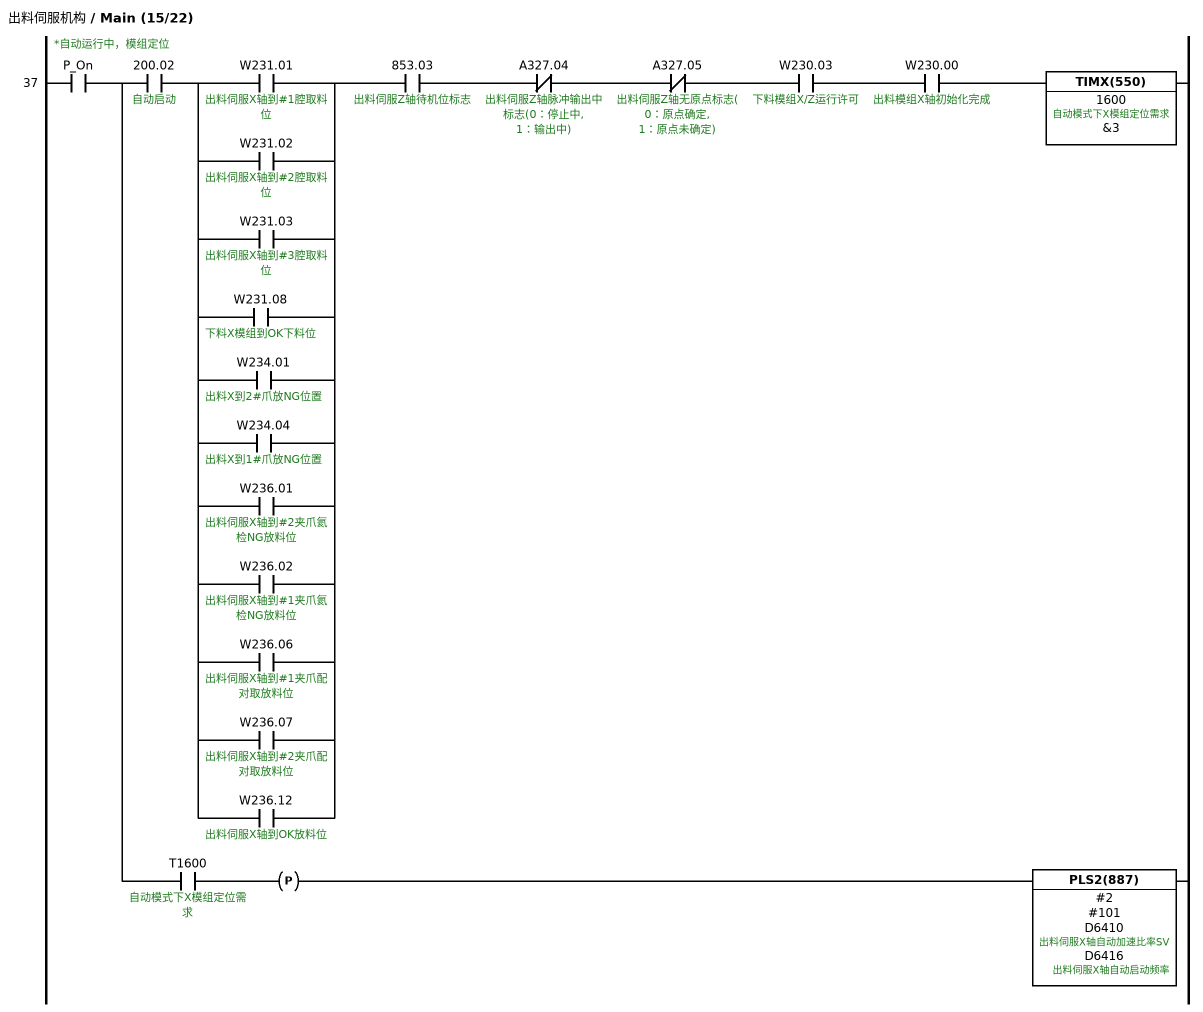
; rung 37: *自动运行中，模组定位
LD P_On
OUT TR0
AND 200.02  ; 自动启动
LD W231.01  ; 出料伺服X轴到#1腔取料位
OR W231.02  ; 出料伺服X轴到#2腔取料位
OR W231.03  ; 出料伺服X轴到#3腔取料位
OR W231.08  ; 下料X模组到OK下料位
OR W234.01  ; 出料X到2#爪放NG位置
OR W234.04  ; 出料X到1#爪放NG位置
OR W236.01  ; 出料伺服X轴到#2夹爪氦检NG放料位
OR W236.02  ; 出料伺服X轴到#1夹爪氦检NG放料位
OR W236.06  ; 出料伺服X轴到#1夹爪配对取放料位
OR W236.07  ; 出料伺服X轴到#2夹爪配对取放料位
OR W236.12  ; 出料伺服X轴到OK放料位
ANDLD
AND 853.03  ; 出料伺服Z轴待机位标志
ANDNOT A327.04  ; 出料伺服Z轴脉冲输出中标志(0：停止中,1：输出中)
ANDNOT A327.05  ; 出料伺服Z轴无原点标志(0：原点确定,1：原点未确定)
AND W230.03  ; 下料模组X/Z运行许可
AND W230.00  ; 出料模组X轴初始化完成
TIMX(550) 1600 &3  ; 自动模式下X模组定位需求
LD TR0
AND T1600  ; 自动模式下X模组定位需求
UP(521)
PLS2(887) #2 #101 D6410 D6416  ; 出料伺服X轴自动加速比率SV, 出料伺服X轴自动启动频率

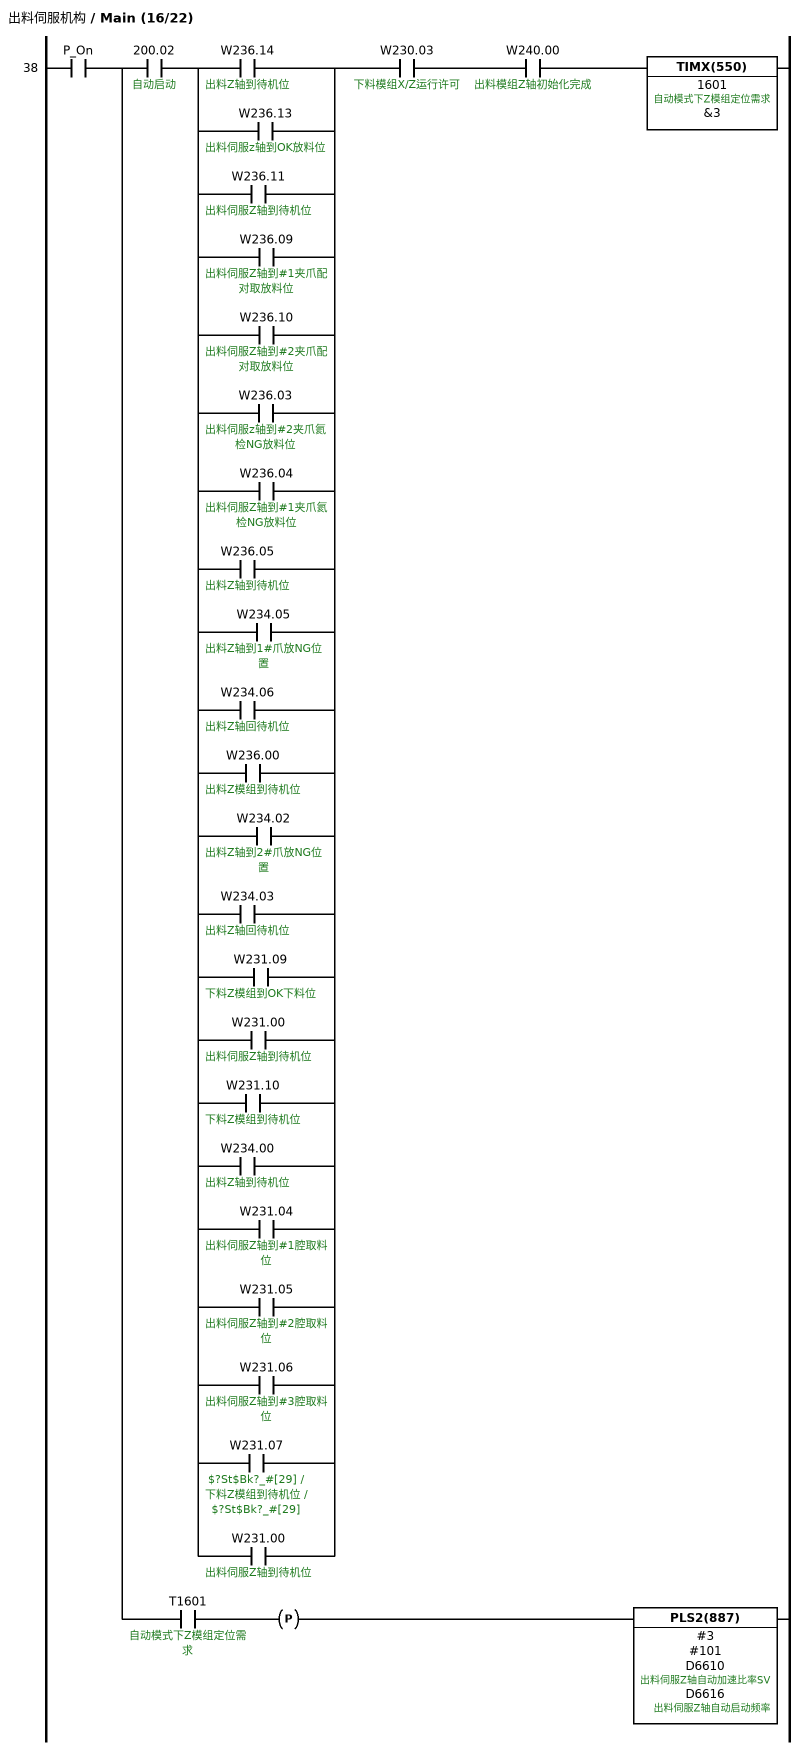
; rung 38
LD P_On
OUT TR0
AND 200.02  ; 自动启动
LD W236.14  ; 出料Z轴到待机位
OR W236.13  ; 出料伺服z轴到OK放料位
OR W236.11  ; 出料伺服Z轴到待机位
OR W236.09  ; 出料伺服Z轴到#1夹爪配对取放料位
OR W236.10  ; 出料伺服Z轴到#2夹爪配对取放料位
OR W236.03  ; 出料伺服z轴到#2夹爪氦检NG放料位
OR W236.04  ; 出料伺服Z轴到#1夹爪氦检NG放料位
OR W236.05  ; 出料Z轴到待机位
OR W234.05  ; 出料Z轴到1#爪放NG位置
OR W234.06  ; 出料Z轴回待机位
OR W236.00  ; 出料Z模组到待机位
OR W234.02  ; 出料Z轴到2#爪放NG位置
OR W234.03  ; 出料Z轴回待机位
OR W231.09  ; 下料Z模组到OK下料位
OR W231.00  ; 出料伺服Z轴到待机位
OR W231.10  ; 下料Z模组到待机位
OR W234.00  ; 出料Z轴到待机位
OR W231.04  ; 出料伺服Z轴到#1腔取料位
OR W231.05  ; 出料伺服Z轴到#2腔取料位
OR W231.06  ; 出料伺服Z轴到#3腔取料位
OR W231.07  ; $?St$Bk?_#[29] / 下料Z模组到待机位 / $?St$Bk?_#[29]
OR W231.00  ; 出料伺服Z轴到待机位
ANDLD
AND W230.03  ; 下料模组X/Z运行许可
AND W240.00  ; 出料模组Z轴初始化完成
TIMX(550) 1601 &3  ; 自动模式下Z模组定位需求
LD TR0
AND T1601  ; 自动模式下Z模组定位需求
UP(521)
PLS2(887) #3 #101 D6610 D6616  ; 出料伺服Z轴自动加速比率SV, 出料伺服Z轴自动启动频率

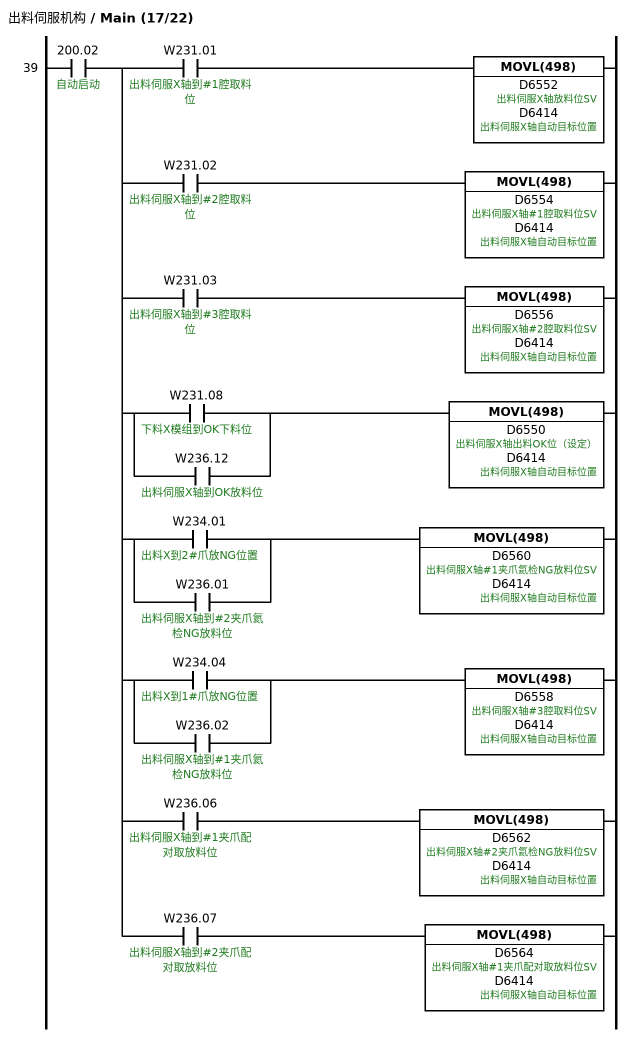
; rung 39
LD 200.02  ; 自动启动
OUT TR0
AND W231.01  ; 出料伺服X轴到#1腔取料位
MOVL(498) D6552 D6414  ; 出料伺服X轴放料位SV, 出料伺服X轴自动目标位置
LD TR0
AND W231.02  ; 出料伺服X轴到#2腔取料位
MOVL(498) D6554 D6414  ; 出料伺服X轴#1腔取料位SV, 出料伺服X轴自动目标位置
LD TR0
AND W231.03  ; 出料伺服X轴到#3腔取料位
MOVL(498) D6556 D6414  ; 出料伺服X轴#2腔取料位SV, 出料伺服X轴自动目标位置
LD TR0
LD W231.08  ; 下料X模组到OK下料位
OR W236.12  ; 出料伺服X轴到OK放料位
ANDLD
MOVL(498) D6550 D6414  ; 出料伺服X轴出料OK位（设定）, 出料伺服X轴自动目标位置
LD TR0
LD W234.01  ; 出料X到2#爪放NG位置
OR W236.01  ; 出料伺服X轴到#2夹爪氦检NG放料位
ANDLD
MOVL(498) D6560 D6414  ; 出料伺服X轴#1夹爪氦检NG放料位SV, 出料伺服X轴自动目标位置
LD TR0
LD W234.04  ; 出料X到1#爪放NG位置
OR W236.02  ; 出料伺服X轴到#1夹爪氦检NG放料位
ANDLD
MOVL(498) D6558 D6414  ; 出料伺服X轴#3腔取料位SV, 出料伺服X轴自动目标位置
LD TR0
AND W236.06  ; 出料伺服X轴到#1夹爪配对取放料位
MOVL(498) D6562 D6414  ; 出料伺服X轴#2夹爪氦检NG放料位SV, 出料伺服X轴自动目标位置
LD TR0
AND W236.07  ; 出料伺服X轴到#2夹爪配对取放料位
MOVL(498) D6564 D6414  ; 出料伺服X轴#1夹爪配对取放料位SV, 出料伺服X轴自动目标位置

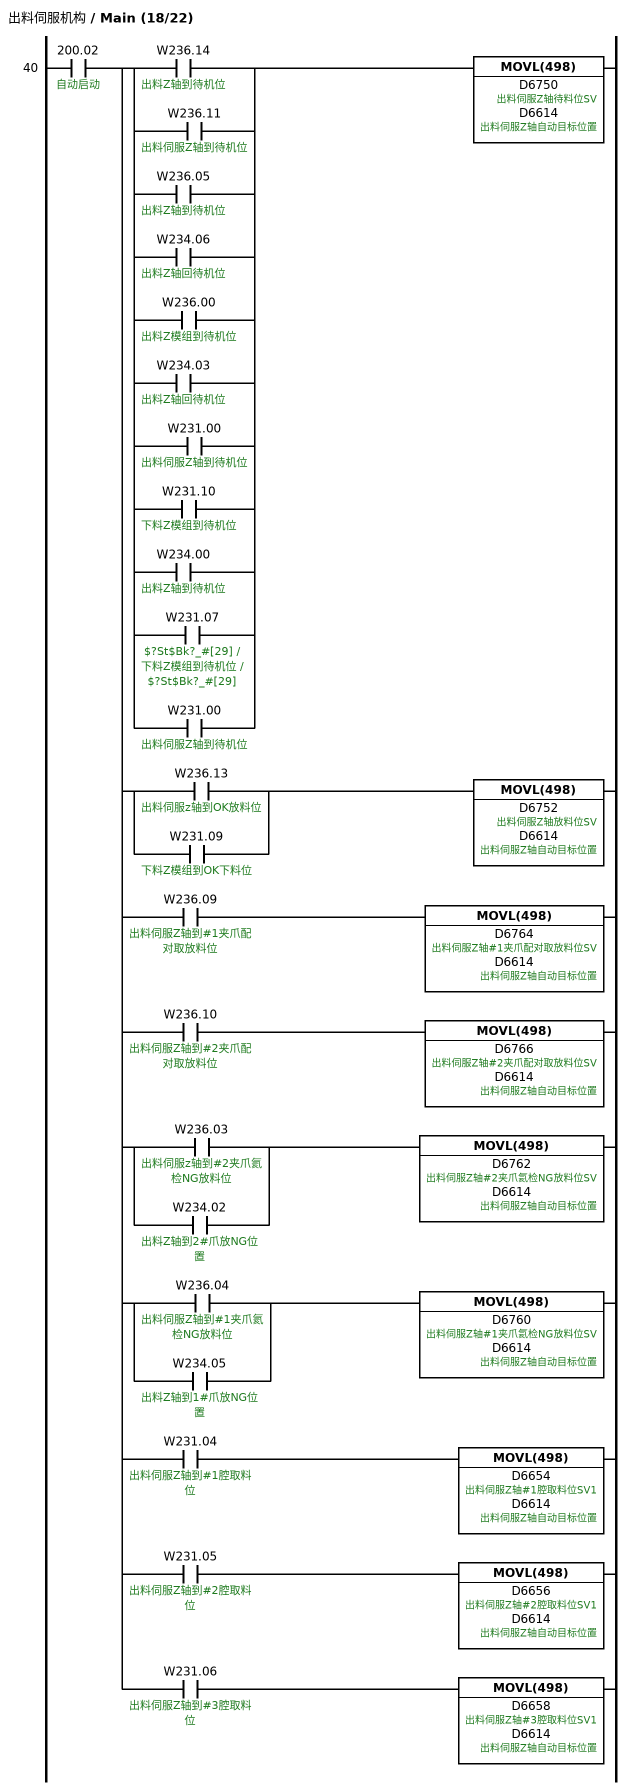
; rung 40
LD 200.02  ; 自动启动
OUT TR0
LD W236.14  ; 出料Z轴到待机位
OR W236.11  ; 出料伺服Z轴到待机位
OR W236.05  ; 出料Z轴到待机位
OR W234.06  ; 出料Z轴回待机位
OR W236.00  ; 出料Z模组到待机位
OR W234.03  ; 出料Z轴回待机位
OR W231.00  ; 出料伺服Z轴到待机位
OR W231.10  ; 下料Z模组到待机位
OR W234.00  ; 出料Z轴到待机位
OR W231.07  ; $?St$Bk?_#[29] / 下料Z模组到待机位 / $?St$Bk?_#[29]
OR W231.00  ; 出料伺服Z轴到待机位
ANDLD
MOVL(498) D6750 D6614  ; 出料伺服Z轴待料位SV, 出料伺服Z轴自动目标位置
LD TR0
LD W236.13  ; 出料伺服z轴到OK放料位
OR W231.09  ; 下料Z模组到OK下料位
ANDLD
MOVL(498) D6752 D6614  ; 出料伺服Z轴放料位SV, 出料伺服Z轴自动目标位置
LD TR0
AND W236.09  ; 出料伺服Z轴到#1夹爪配对取放料位
MOVL(498) D6764 D6614  ; 出料伺服Z轴#1夹爪配对取放料位SV, 出料伺服Z轴自动目标位置
LD TR0
AND W236.10  ; 出料伺服Z轴到#2夹爪配对取放料位
MOVL(498) D6766 D6614  ; 出料伺服Z轴#2夹爪配对取放料位SV, 出料伺服Z轴自动目标位置
LD TR0
LD W236.03  ; 出料伺服z轴到#2夹爪氦检NG放料位
OR W234.02  ; 出料Z轴到2#爪放NG位置
ANDLD
MOVL(498) D6762 D6614  ; 出料伺服Z轴#2夹爪氦检NG放料位SV, 出料伺服Z轴自动目标位置
LD TR0
LD W236.04  ; 出料伺服Z轴到#1夹爪氦检NG放料位
OR W234.05  ; 出料Z轴到1#爪放NG位置
ANDLD
MOVL(498) D6760 D6614  ; 出料伺服Z轴#1夹爪氦检NG放料位SV, 出料伺服Z轴自动目标位置
LD TR0
AND W231.04  ; 出料伺服Z轴到#1腔取料位
MOVL(498) D6654 D6614  ; 出料伺服Z轴#1腔取料位SV1, 出料伺服Z轴自动目标位置
LD TR0
AND W231.05  ; 出料伺服Z轴到#2腔取料位
MOVL(498) D6656 D6614  ; 出料伺服Z轴#2腔取料位SV1, 出料伺服Z轴自动目标位置
LD TR0
AND W231.06  ; 出料伺服Z轴到#3腔取料位
MOVL(498) D6658 D6614  ; 出料伺服Z轴#3腔取料位SV1, 出料伺服Z轴自动目标位置

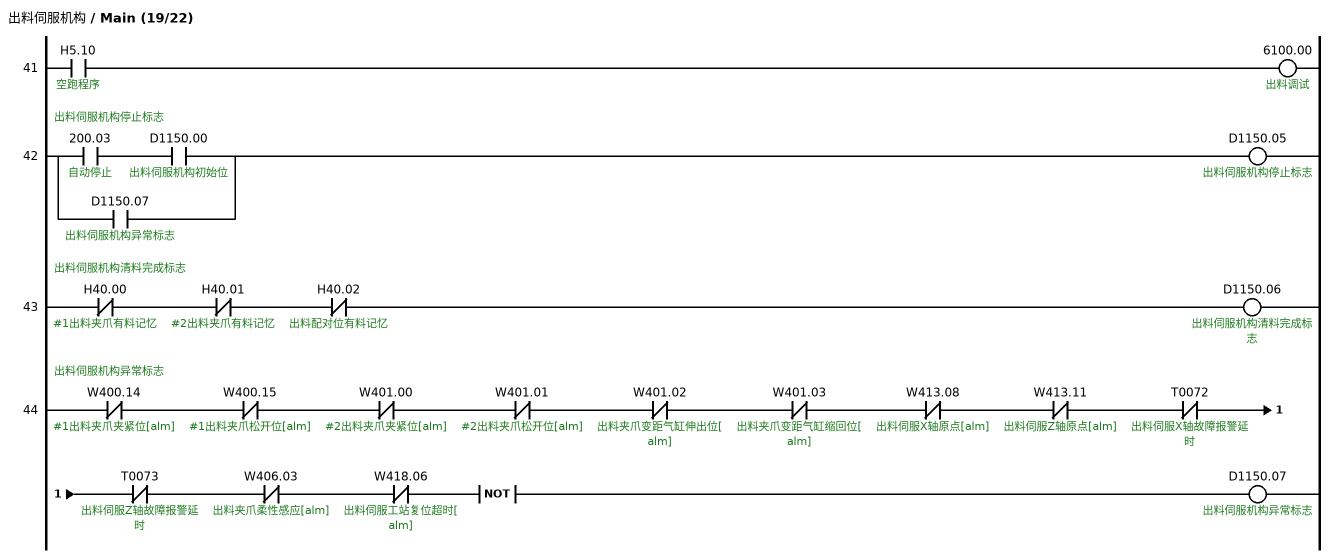
; rung 41
LD H5.10  ; 空跑程序
OUT 6100.00  ; 出料调试
; rung 42: 出料伺服机构停止标志
LD 200.03  ; 自动停止
AND D1150.00  ; 出料伺服机构初始位
OR D1150.07  ; 出料伺服机构异常标志
OUT D1150.05  ; 出料伺服机构停止标志
; rung 43: 出料伺服机构清料完成标志
LDNOT H40.00  ; #1出料夹爪有料记忆
ANDNOT H40.01  ; #2出料夹爪有料记忆
ANDNOT H40.02  ; 出料配对位有料记忆
OUT D1150.06  ; 出料伺服机构清料完成标志
; rung 44: 出料伺服机构异常标志
LDNOT W400.14  ; #1出料夹爪夹紧位[alm]
ANDNOT W400.15  ; #1出料夹爪松开位[alm]
ANDNOT W401.00  ; #2出料夹爪夹紧位[alm]
ANDNOT W401.01  ; #2出料夹爪松开位[alm]
ANDNOT W401.02  ; 出料夹爪变距气缸伸出位[alm]
ANDNOT W401.03  ; 出料夹爪变距气缸缩回位[alm]
ANDNOT W413.08  ; 出料伺服X轴原点[alm]
ANDNOT W413.11  ; 出料伺服Z轴原点[alm]
ANDNOT T0072  ; 出料伺服X轴故障报警延时
ANDNOT T0073  ; 出料伺服Z轴故障报警延时
ANDNOT W406.03  ; 出料夹爪柔性感应[alm]
ANDNOT W418.06  ; 出料伺服工站复位超时[alm]
NOT(520)
OUT D1150.07  ; 出料伺服机构异常标志

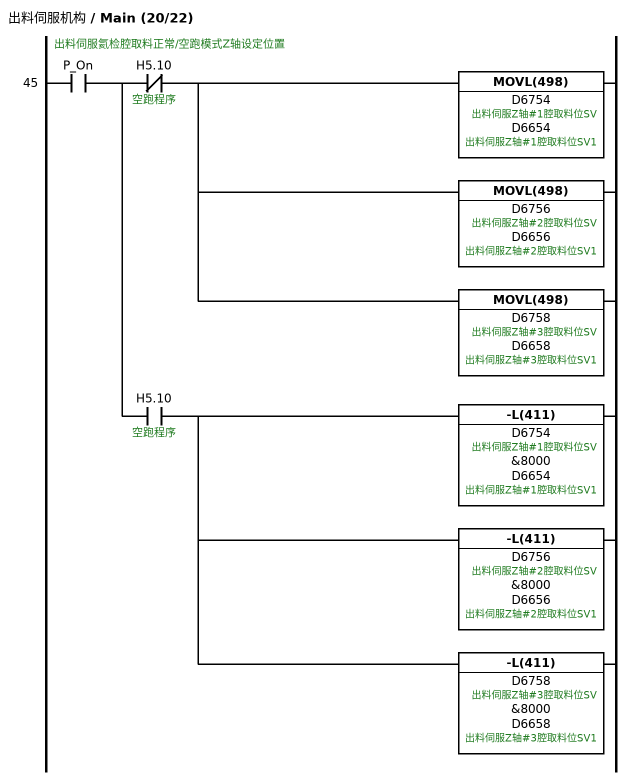
; rung 45: 出料伺服氦检腔取料正常/空跑模式Z轴设定位置
LD P_On
OUT TR0
ANDNOT H5.10  ; 空跑程序
MOVL(498) D6754 D6654  ; 出料伺服Z轴#1腔取料位SV, 出料伺服Z轴#1腔取料位SV1
MOVL(498) D6756 D6656  ; 出料伺服Z轴#2腔取料位SV, 出料伺服Z轴#2腔取料位SV1
MOVL(498) D6758 D6658  ; 出料伺服Z轴#3腔取料位SV, 出料伺服Z轴#3腔取料位SV1
LD TR0
AND H5.10  ; 空跑程序
-L(411) D6754 &8000 D6654  ; 出料伺服Z轴#1腔取料位SV, 出料伺服Z轴#1腔取料位SV1
-L(411) D6756 &8000 D6656  ; 出料伺服Z轴#2腔取料位SV, 出料伺服Z轴#2腔取料位SV1
-L(411) D6758 &8000 D6658  ; 出料伺服Z轴#3腔取料位SV, 出料伺服Z轴#3腔取料位SV1

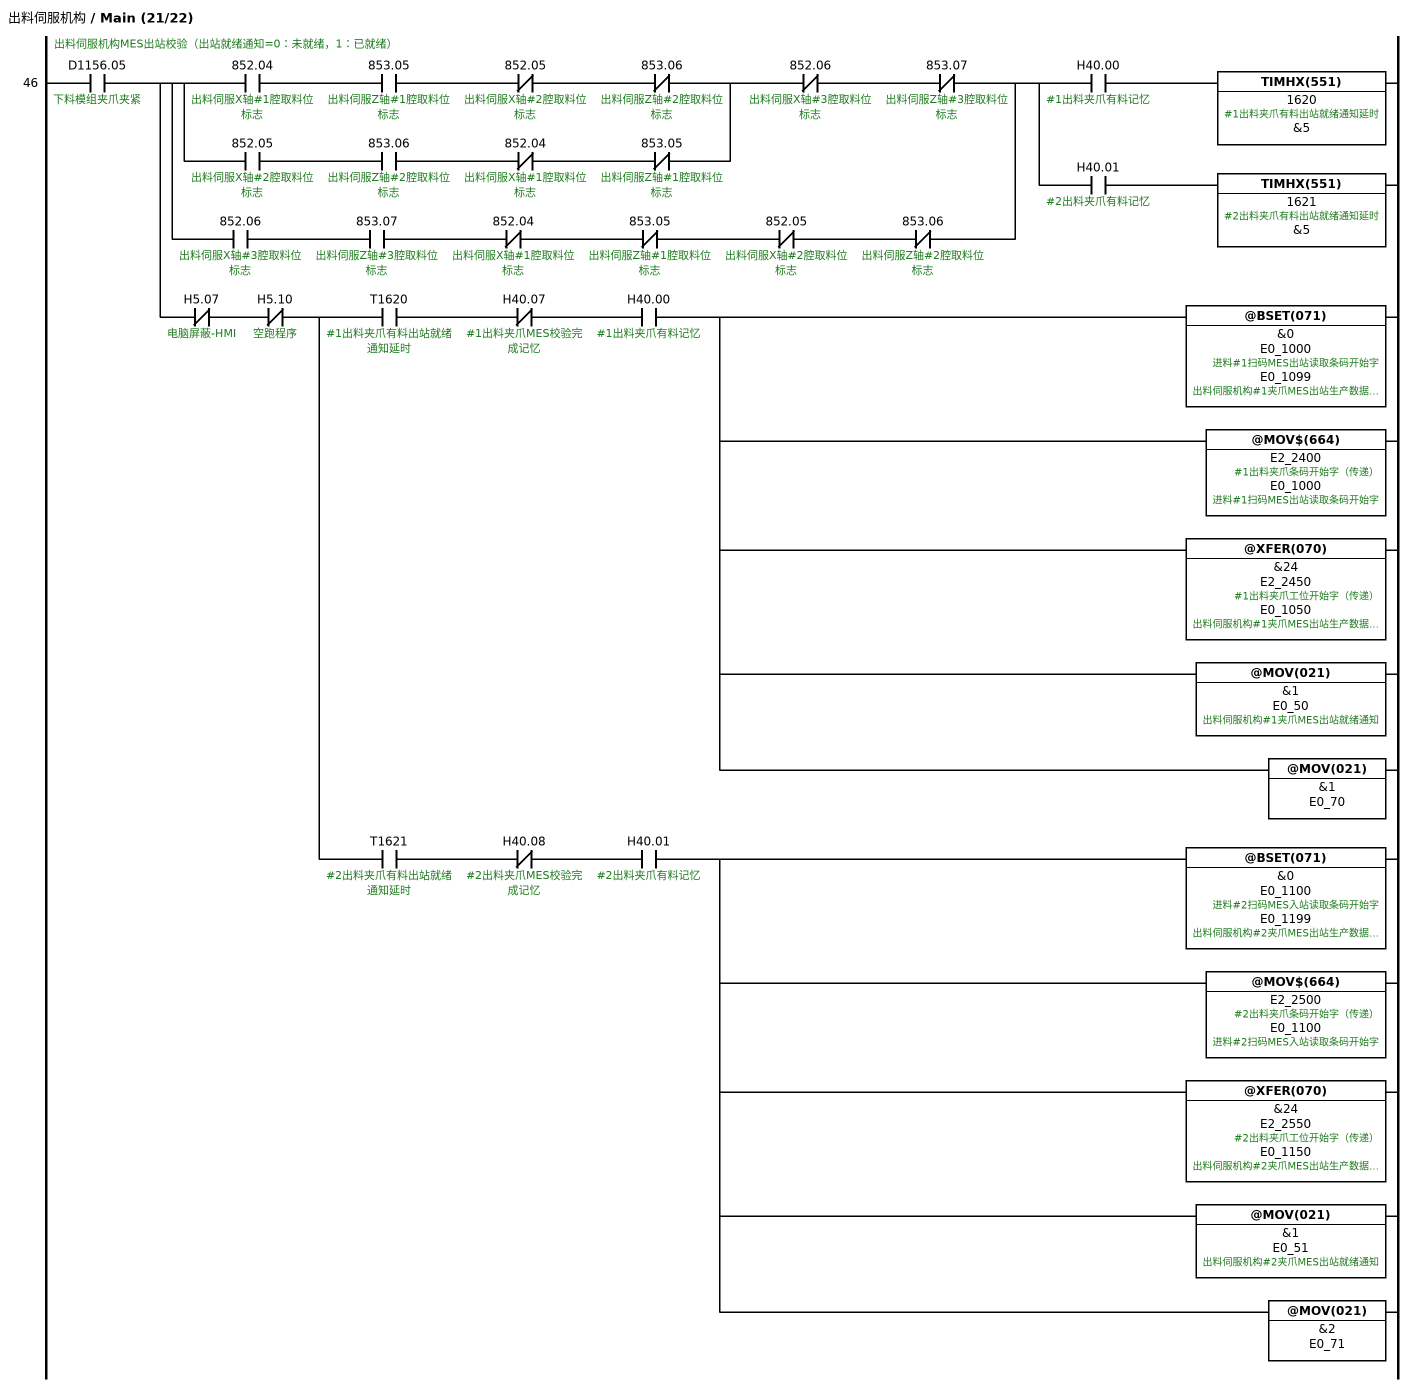
; rung 46: 出料伺服机构MES出站校验（出站就绪通知=0：未就绪，1：已就绪）
LD D1156.05  ; 下料模组夹爪夹紧
OUT TR0
LD 852.04  ; 出料伺服X轴#1腔取料位标志
AND 853.05  ; 出料伺服Z轴#1腔取料位标志
ANDNOT 852.05  ; 出料伺服X轴#2腔取料位标志
ANDNOT 853.06  ; 出料伺服Z轴#2腔取料位标志
LD 852.05  ; 出料伺服X轴#2腔取料位标志
AND 853.06  ; 出料伺服Z轴#2腔取料位标志
ANDNOT 852.04  ; 出料伺服X轴#1腔取料位标志
ANDNOT 853.05  ; 出料伺服Z轴#1腔取料位标志
ORLD
ANDNOT 852.06  ; 出料伺服X轴#3腔取料位标志
ANDNOT 853.07  ; 出料伺服Z轴#3腔取料位标志
LD 852.06  ; 出料伺服X轴#3腔取料位标志
AND 853.07  ; 出料伺服Z轴#3腔取料位标志
ANDNOT 852.04  ; 出料伺服X轴#1腔取料位标志
ANDNOT 853.05  ; 出料伺服Z轴#1腔取料位标志
ANDNOT 852.05  ; 出料伺服X轴#2腔取料位标志
ANDNOT 853.06  ; 出料伺服Z轴#2腔取料位标志
ORLD
ANDLD
OUT TR1
AND H40.00  ; #1出料夹爪有料记忆
TIMHX(551) 1620 &5  ; #1出料夹爪有料出站就绪通知延时
LD TR1
AND H40.01  ; #2出料夹爪有料记忆
TIMHX(551) 1621 &5  ; #2出料夹爪有料出站就绪通知延时
LD TR0
ANDNOT H5.07  ; 电脑屏蔽-HMI
ANDNOT H5.10  ; 空跑程序
OUT TR0
AND T1620  ; #1出料夹爪有料出站就绪通知延时
ANDNOT H40.07  ; #1出料夹爪MES校验完成记忆
AND H40.00  ; #1出料夹爪有料记忆
@BSET(071) &0 E0_1000 E0_1099  ; 进料#1扫码MES出站读取条码开始字, 出料伺服机构#1夹爪MES出站生产数据结束字
@MOV$(664) E2_2400 E0_1000  ; #1出料夹爪条码开始字（传递）, 进料#1扫码MES出站读取条码开始字
@XFER(070) &24 E2_2450 E0_1050  ; #1出料夹爪工位开始字（传递）, 出料伺服机构#1夹爪MES出站生产数据开始字
@MOV(021) &1 E0_50  ; 出料伺服机构#1夹爪MES出站就绪通知
@MOV(021) &1 E0_70
LD TR0
AND T1621  ; #2出料夹爪有料出站就绪通知延时
ANDNOT H40.08  ; #2出料夹爪MES校验完成记忆
AND H40.01  ; #2出料夹爪有料记忆
@BSET(071) &0 E0_1100 E0_1199  ; 进料#2扫码MES入站读取条码开始字, 出料伺服机构#2夹爪MES出站生产数据结束字
@MOV$(664) E2_2500 E0_1100  ; #2出料夹爪条码开始字（传递）, 进料#2扫码MES入站读取条码开始字
@XFER(070) &24 E2_2550 E0_1150  ; #2出料夹爪工位开始字（传递）, 出料伺服机构#2夹爪MES出站生产数据开始字
@MOV(021) &1 E0_51  ; 出料伺服机构#2夹爪MES出站就绪通知
@MOV(021) &2 E0_71

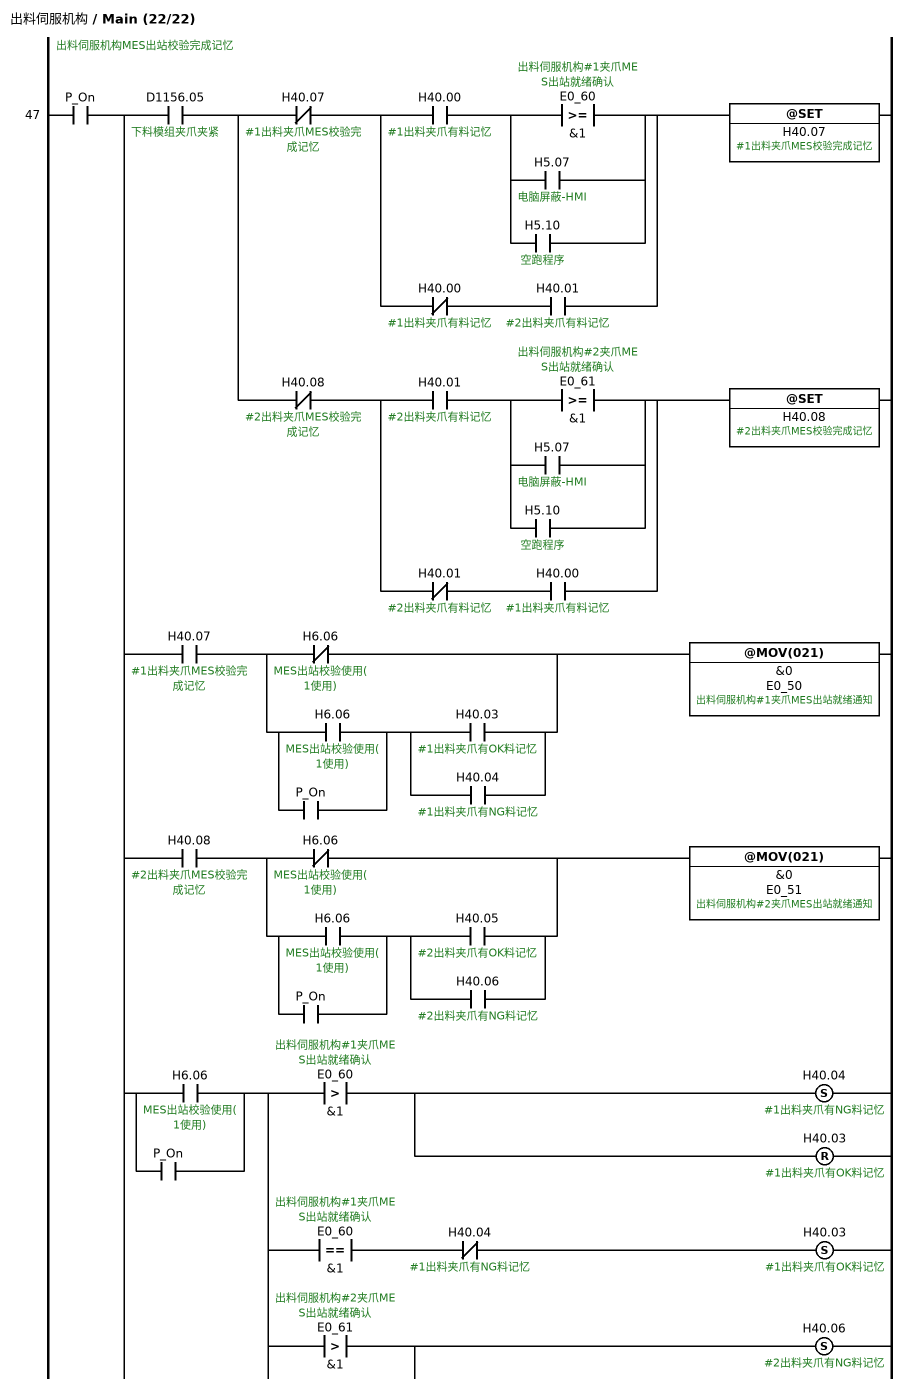

